C05475=1188.740,321.478,-72.281,-176.478,7.828,148.484
C05476=1188.743,321.230,-72.249,-176.480,7.825,148.484
C05477=1188.748,320.982,-72.218,-176.482,7.823,148.484
C05478=1188.752,320.734,-72.187,-176.485,7.820,148.484
C05479=1188.756,320.486,-72.156,-176.487,7.816,148.484
C05480=1188.760,320.238,-72.124,-176.490,7.813,148.484
C05481=1188.765,319.990,-72.093,-176.492,7.810,148.484
C05482=1188.769,319.743,-72.062,-176.495,7.807,148.484
C05483=1188.773,319.494,-72.031,-176.497,7.805,148.484
C05484=1188.777,319.246,-72.000,-176.499,7.802,148.484
C05485=1188.780,318.999,-71.969,-176.502,7.799,148.484
C05486=1188.785,318.751,-71.938,-176.504,7.795,148.484
C05487=1188.789,318.503,-71.906,-176.507,7.792,148.484
C05488=1188.793,318.255,-71.875,-176.509,7.789,148.484
C05489=1188.797,318.006,-71.844,-176.512,7.786,148.483
C05490=1188.802,317.759,-71.813,-176.514,7.784,148.483
C05491=1188.806,317.511,-71.782,-176.516,7.781,148.483
C05492=1188.810,317.262,-71.751,-176.519,7.777,148.483
C05493=1188.815,317.014,-71.720,-176.521,7.774,148.483
C05494=1188.819,316.766,-71.688,-176.524,7.771,148.483
C05495=1188.823,316.518,-71.657,-176.526,7.768,148.483
C05496=1188.827,316.271,-71.627,-176.529,7.766,148.483
C05497=1188.831,316.022,-71.596,-176.531,7.763,148.483
C05498=1188.835,315.775,-71.565,-176.533,7.759,148.483
C05499=1188.840,315.527,-71.534,-176.536,7.756,148.483
C05500=1188.844,315.278,-71.503,-176.539,7.753,148.483
C05501=1188.849,315.030,-71.472,-176.541,7.750,148.483
C05502=1188.853,314.753,-71.437,-176.544,7.747,148.483
C05503=1188.858,314.477,-71.404,-176.547,7.744,148.483
C05504=1188.862,314.201,-71.369,-176.549,7.741,148.483
C05505=1188.867,313.924,-71.334,-176.553,7.737,148.483
C05506=1188.871,313.676,-71.304,-176.554,7.735,148.483
C05507=1188.876,313.428,-71.273,-176.557,7.732,148.483
C05508=1188.880,313.180,-71.242,-176.560,7.729,148.483
C05509=1188.884,312.932,-71.211,-176.562,7.725,148.482
C05510=1188.888,312.684,-71.181,-176.565,7.722,148.482
C05511=1188.893,312.436,-71.150,-176.567,7.719,148.482
C05512=1188.897,312.187,-71.119,-176.569,7.717,148.482
C05513=1188.901,311.939,-71.088,-176.572,7.714,148.482
C05514=1188.905,311.692,-71.058,-176.574,7.711,148.482
C05515=1188.909,311.443,-71.027,-176.577,7.708,148.482
C05516=1188.914,311.195,-70.996,-176.579,7.705,148.482
C05517=1188.918,310.947,-70.966,-176.581,7.702,148.482
C05518=1188.922,310.699,-70.935,-176.584,7.699,148.482
C05519=1188.926,310.451,-70.904,-176.587,7.696,148.482
C05520=1188.930,310.203,-70.874,-176.589,7.693,148.482
C05521=1188.935,309.955,-70.843,-176.592,7.690,148.482
C05522=1188.939,309.707,-70.812,-176.594,7.688,148.482
C05523=1188.943,309.459,-70.782,-176.597,7.685,148.482
C05524=1188.948,309.210,-70.752,-176.599,7.682,148.482
C05525=1188.952,308.962,-70.721,-176.602,7.679,148.482
C05526=1188.956,308.715,-70.691,-176.604,7.676,148.482
C05527=1188.960,308.466,-70.660,-176.607,7.673,148.482
C05528=1188.964,308.218,-70.630,-176.609,7.670,148.482
C05529=1188.969,307.970,-70.599,-176.611,7.667,148.482
C05530=1188.973,307.722,-70.569,-176.614,7.664,148.482
C05531=1188.977,307.474,-70.539,-176.617,7.661,148.482
C05532=1188.981,307.226,-70.507,-176.620,7.658,148.482
C05533=1188.985,306.978,-70.477,-176.622,7.656,148.482
C05534=1188.990,306.729,-70.447,-176.624,7.653,148.482
C05535=1188.995,306.481,-70.416,-176.627,7.650,148.482
C05536=1188.999,306.234,-70.386,-176.629,7.647,148.482
C05537=1189.003,305.986,-70.356,-176.632,7.644,148.482
C05538=1189.007,305.737,-70.326,-176.634,7.641,148.482
C05539=1189.011,305.489,-70.295,-176.637,7.638,148.482
C05540=1189.015,305.241,-70.265,-176.639,7.635,148.482
C05541=1189.020,304.993,-70.235,-176.642,7.632,148.482
C05542=1189.024,304.745,-70.205,-176.644,7.630,148.482
C05543=1189.029,304.496,-70.175,-176.647,7.627,148.482
C05544=1189.032,304.248,-70.144,-176.649,7.624,148.482
C05545=1189.037,304.000,-70.113,-176.652,7.621,148.482
C05546=1189.041,303.752,-70.084,-176.654,7.618,148.482
C05547=1189.045,303.504,-70.054,-176.657,7.615,148.482
C05548=1189.050,303.256,-70.024,-176.659,7.612,148.482
C05549=1189.054,303.008,-69.993,-176.662,7.609,148.482
C05550=1189.059,302.759,-69.963,-176.665,7.606,148.482
C05551=1189.063,302.512,-69.933,-176.667,7.604,148.482
C05552=1189.068,302.263,-69.903,-176.669,7.601,148.482
C05553=1189.071,302.015,-69.873,-176.672,7.598,148.482
C05554=1189.075,301.767,-69.843,-176.675,7.595,148.482
C05555=1189.080,301.519,-69.812,-176.677,7.592,148.482
C05556=1189.084,301.270,-69.783,-176.679,7.590,148.482
C05557=1189.088,301.023,-69.753,-176.682,7.587,148.482
C05558=1189.093,300.774,-69.723,-176.685,7.584,148.482
C05559=1189.096,300.526,-69.693,-176.688,7.581,148.482
C05560=1189.101,300.278,-69.662,-176.689,7.578,148.482
C05561=1189.106,300.030,-69.633,-176.692,7.575,148.482
C05562=1189.109,299.782,-69.603,-176.695,7.572,148.482
C05563=1189.114,299.534,-69.573,-176.697,7.569,148.482
C05564=1189.118,299.286,-69.543,-176.700,7.567,148.482
C05565=1189.122,299.037,-69.513,-176.702,7.564,148.482
C05566=1189.127,298.789,-69.484,-176.705,7.561,148.482
C05567=1189.131,298.541,-69.453,-176.708,7.558,148.482
C05568=1189.135,298.293,-69.424,-176.710,7.555,148.482
C05569=1189.140,298.045,-69.394,-176.712,7.552,148.482
C05570=1189.144,297.796,-69.365,-176.715,7.549,148.482
C05571=1189.148,297.548,-69.334,-176.717,7.546,148.482
C05572=1189.153,297.300,-69.304,-176.720,7.543,148.482
C05573=1189.157,297.052,-69.275,-176.722,7.541,148.482
C05574=1189.161,296.804,-69.245,-176.725,7.538,148.482
C05575=1189.165,296.556,-69.215,-176.728,7.535,148.482
C05576=1189.170,296.307,-69.185,-176.730,7.532,148.482
C05577=1189.174,296.059,-69.156,-176.733,7.530,148.482
C05578=1189.178,295.811,-69.126,-176.735,7.527,148.482
C05579=1189.182,295.563,-69.097,-176.738,7.524,148.482
C05580=1189.186,295.315,-69.067,-176.740,7.522,148.482
C05581=1189.191,295.066,-69.037,-176.743,7.519,148.482
C05582=1189.195,294.818,-69.007,-176.746,7.516,148.482
C05583=1189.199,294.570,-68.978,-176.748,7.513,148.482
C05584=1189.204,294.322,-68.948,-176.750,7.510,148.482
C05585=1189.208,294.073,-68.919,-176.753,7.507,148.482
C05586=1189.212,293.825,-68.889,-176.755,7.504,148.482
C05587=1189.216,293.577,-68.860,-176.758,7.501,148.482
C05588=1189.220,293.329,-68.831,-176.760,7.499,148.482
C05589=1189.225,293.080,-68.800,-176.763,7.496,148.482
C05590=1189.229,292.832,-68.771,-176.766,7.493,148.482
C05591=1189.234,292.583,-68.742,-176.768,7.490,148.482
C05592=1189.238,292.336,-68.712,-176.771,7.488,148.482
C05593=1189.243,292.088,-68.683,-176.773,7.485,148.482
C05594=1189.247,291.839,-68.654,-176.776,7.482,148.482
C05595=1189.251,291.591,-68.624,-176.778,7.480,148.482
C05596=1189.255,291.343,-68.595,-176.781,7.477,148.482
C05597=1189.259,291.094,-68.565,-176.784,7.474,148.482
C05598=1189.263,290.846,-68.536,-176.786,7.471,148.482
C05599=1189.268,290.598,-68.506,-176.788,7.469,148.483
C05600=1189.272,290.350,-68.477,-176.791,7.466,148.483
C05601=1189.277,290.102,-68.448,-176.794,7.463,148.483
C05602=1189.281,289.854,-68.418,-176.796,7.461,148.483
C05603=1189.285,289.605,-68.390,-176.799,7.458,148.483
C05604=1189.289,289.357,-68.360,-176.801,7.455,148.483
C05605=1189.294,289.108,-68.331,-176.804,7.452,148.483
C05606=1189.298,288.835,-68.298,-176.807,7.449,148.483
C05607=1189.303,288.559,-68.266,-176.810,7.446,148.483
C05608=1189.308,288.285,-68.234,-176.812,7.443,148.483
C05609=1189.313,288.011,-68.201,-176.815,7.440,148.483
C05610=1189.318,287.762,-68.172,-176.818,7.437,148.483
C05611=1189.321,287.514,-68.144,-176.820,7.435,148.483
C05612=1189.325,287.266,-68.114,-176.823,7.432,148.483
C05613=1189.330,287.018,-68.085,-176.826,7.429,148.483
C05614=1189.334,286.769,-68.056,-176.828,7.427,148.483
C05615=1189.339,286.521,-68.027,-176.831,7.424,148.483
C05616=1189.343,286.273,-67.997,-176.833,7.421,148.483
C05617=1189.347,286.024,-67.969,-176.836,7.418,148.483
C05618=1189.352,285.776,-67.940,-176.838,7.415,148.483
C05619=1189.356,285.528,-67.911,-176.841,7.412,148.483
C05620=1189.360,285.280,-67.882,-176.844,7.409,148.483
C05621=1189.364,285.031,-67.852,-176.846,7.407,148.484
C05622=1189.369,284.784,-67.823,-176.849,7.404,148.484
C05623=1189.374,284.535,-67.795,-176.851,7.401,148.484
C05624=1189.378,284.287,-67.765,-176.853,7.399,148.484
C05625=1189.381,284.038,-67.737,-176.856,7.396,148.484
C05626=1189.386,283.790,-67.708,-176.859,7.393,148.484
C05627=1189.391,283.541,-67.679,-176.861,7.391,148.484
C05628=1189.395,283.293,-67.650,-176.864,7.388,148.484
C05629=1189.399,283.044,-67.621,-176.866,7.385,148.484
C05630=1189.403,282.797,-67.593,-176.869,7.383,148.484
C05631=1189.408,282.548,-67.564,-176.872,7.380,148.484
C05632=1189.412,282.300,-67.534,-176.874,7.377,148.484
C05633=1189.417,282.052,-67.506,-176.877,7.375,148.484
C05634=1189.421,281.804,-67.477,-176.879,7.372,148.484
C05635=1189.425,281.555,-67.448,-176.882,7.369,148.484
C05636=1189.430,281.307,-67.419,-176.884,7.367,148.484
C05637=1189.434,281.059,-67.391,-176.887,7.364,148.485
C05638=1189.438,280.810,-67.362,-176.890,7.361,148.485
C05639=1189.443,280.562,-67.333,-176.892,7.359,148.485
C05640=1189.447,280.314,-67.305,-176.895,7.356,148.485
C05641=1189.451,280.065,-67.276,-176.898,7.353,148.485
C05642=1189.456,279.817,-67.247,-176.900,7.351,148.485
C05643=1189.460,279.569,-67.219,-176.903,7.348,148.485
C05644=1189.464,279.320,-67.190,-176.905,7.345,148.485
C05645=1189.469,279.072,-67.161,-176.907,7.343,148.485
C05646=1189.473,278.824,-67.133,-176.910,7.340,148.485
C05647=1189.477,278.575,-67.104,-176.913,7.337,148.485
C05648=1189.482,278.327,-67.075,-176.915,7.334,148.485
C05649=1189.486,278.079,-67.047,-176.918,7.331,148.485
C05650=1189.490,277.831,-67.018,-176.920,7.330,148.486
C05651=1189.494,277.582,-66.990,-176.923,7.327,148.486
C05652=1189.499,277.334,-66.961,-176.926,7.324,148.486
C05653=1189.503,277.086,-66.934,-176.928,7.321,148.486
C05654=1189.508,276.837,-66.905,-176.931,7.318,148.486
C05655=1189.512,276.589,-66.876,-176.933,7.315,148.486
C05656=1189.516,276.341,-66.848,-176.936,7.313,148.486
C05657=1189.521,276.092,-66.819,-176.938,7.310,148.486
C05658=1189.525,275.844,-66.791,-176.941,7.308,148.486
C05659=1189.529,275.595,-66.762,-176.944,7.305,148.486
C05660=1189.534,275.347,-66.735,-176.946,7.302,148.486
C05661=1189.538,275.099,-66.705,-176.948,7.300,148.486
C05662=1189.542,274.851,-66.677,-176.951,7.297,148.486
C05663=1189.547,274.602,-66.649,-176.954,7.294,148.487
C05664=1189.551,274.354,-66.620,-176.956,7.292,148.487
C05665=1189.556,274.105,-66.592,-176.959,7.289,148.487
C05666=1189.559,273.857,-66.564,-176.962,7.286,148.487
C05667=1189.564,273.609,-66.536,-176.964,7.284,148.487
C05668=1189.568,273.360,-66.507,-176.967,7.281,148.487
C05669=1189.573,273.112,-66.480,-176.969,7.279,148.487
C05670=1189.577,272.863,-66.451,-176.972,7.276,148.487
C05671=1189.581,272.615,-66.423,-176.975,7.273,148.487
C05672=1189.586,272.367,-66.394,-176.977,7.271,148.487
C05673=1189.590,272.119,-66.367,-176.980,7.268,148.488
C05674=1189.594,271.870,-66.338,-176.982,7.266,148.488
C05675=1189.599,271.622,-66.310,-176.985,7.263,148.488
C05676=1189.603,271.373,-66.282,-176.988,7.260,148.488
C05677=1189.608,271.125,-66.254,-176.990,7.258,148.488
C05678=1189.612,270.877,-66.225,-176.993,7.255,148.488
C05679=1189.616,270.629,-66.198,-176.995,7.253,148.488
C05680=1189.621,270.380,-66.169,-176.998,7.250,148.488
C05681=1189.625,270.131,-66.142,-177.000,7.247,148.488
C05682=1189.630,269.883,-66.114,-177.003,7.245,148.488
C05683=1189.634,269.635,-66.085,-177.006,7.242,148.489
C05684=1189.638,269.387,-66.058,-177.008,7.240,148.489
C05685=1189.642,269.138,-66.029,-177.011,7.237,148.489
C05686=1189.647,268.890,-66.001,-177.013,7.235,148.489
C05687=1189.651,268.641,-65.974,-177.016,7.232,148.489
C05688=1189.656,268.393,-65.946,-177.019,7.229,148.489
C05689=1189.661,268.145,-65.917,-177.021,7.227,148.489
C05690=1189.664,267.896,-65.889,-177.024,7.224,148.489
C05691=1189.669,267.648,-65.862,-177.026,7.222,148.489
C05692=1189.673,267.399,-65.834,-177.029,7.219,148.490
C05693=1189.678,267.151,-65.806,-177.031,7.217,148.490
C05694=1189.682,266.903,-65.778,-177.034,7.214,148.490
C05695=1189.686,266.654,-65.751,-177.036,7.211,148.490
C05696=1189.691,266.406,-65.723,-177.039,7.209,148.490
C05697=1189.694,266.157,-65.695,-177.042,7.206,148.490
C05698=1189.700,265.908,-65.667,-177.044,7.204,148.490
C05699=1189.704,265.661,-65.639,-177.047,7.201,148.490
C05700=1189.708,265.412,-65.611,-177.049,7.199,148.490
C05701=1189.713,265.163,-65.584,-177.052,7.196,148.491
C05702=1189.717,264.916,-65.556,-177.055,7.193,148.491
C05703=1189.722,264.666,-65.528,-177.057,7.191,148.491
C05704=1189.726,264.418,-65.500,-177.060,7.188,148.491
C05705=1189.730,264.170,-65.473,-177.062,7.186,148.491
C05706=1189.735,263.921,-65.445,-177.065,7.183,148.491
C05707=1189.739,263.673,-65.417,-177.067,7.181,148.491
C05708=1189.744,263.425,-65.390,-177.070,7.178,148.491
C05709=1189.747,263.176,-65.362,-177.072,7.176,148.491
C05710=1189.753,262.904,-65.332,-177.075,7.173,148.492
C05711=1189.757,262.630,-65.301,-177.078,7.171,148.492
C05712=1189.762,262.358,-65.271,-177.081,7.168,148.492
C05713=1189.766,262.085,-65.241,-177.084,7.165,148.492
C05714=1189.772,261.836,-65.213,-177.086,7.163,148.492
C05715=1189.776,261.587,-65.186,-177.089,7.160,148.492
C05716=1189.781,261.339,-65.158,-177.091,7.158,148.492
C05717=1189.785,261.090,-65.131,-177.095,7.155,148.493
C05718=1189.789,260.842,-65.103,-177.097,7.152,148.493
C05719=1189.794,260.594,-65.076,-177.099,7.150,148.493
C05720=1189.798,260.345,-65.048,-177.102,7.147,148.493
C05721=1189.802,260.097,-65.021,-177.105,7.145,148.493
C05722=1189.807,259.848,-64.994,-177.108,7.142,148.493
C05723=1189.811,259.600,-64.966,-177.110,7.140,148.493
C05724=1189.815,259.351,-64.939,-177.113,7.137,148.493
C05725=1189.820,259.103,-64.912,-177.115,7.135,148.494
C05726=1189.824,258.855,-64.884,-177.118,7.132,148.494
C05727=1189.829,258.606,-64.857,-177.120,7.130,148.494
C05728=1189.834,258.358,-64.830,-177.123,7.127,148.494
C05729=1189.838,258.109,-64.802,-177.125,7.125,148.494
C05730=1189.842,257.861,-64.774,-177.128,7.122,148.494
C05731=1189.847,257.612,-64.747,-177.131,7.120,148.494
C05732=1189.851,257.364,-64.721,-177.133,7.117,148.494
C05733=1189.855,257.115,-64.693,-177.136,7.115,148.495
C05734=1189.859,256.867,-64.666,-177.139,7.112,148.495
C05735=1189.864,256.619,-64.639,-177.141,7.110,148.495
C05736=1189.868,256.370,-64.612,-177.144,7.107,148.495
C05737=1189.873,256.122,-64.585,-177.146,7.105,148.495
C05738=1189.878,255.873,-64.557,-177.149,7.102,148.495
C05739=1189.881,255.624,-64.529,-177.151,7.100,148.495
C05740=1189.886,255.376,-64.502,-177.154,7.098,148.496
C05741=1189.890,255.128,-64.476,-177.156,7.095,148.496
C05742=1189.895,254.879,-64.449,-177.159,7.092,148.496
C05743=1189.899,254.631,-64.422,-177.162,7.091,148.496
C05744=1189.904,254.382,-64.395,-177.165,7.088,148.496
C05745=1189.908,254.133,-64.367,-177.167,7.086,148.497
C05746=1189.913,253.885,-64.340,-177.170,7.083,148.497
C05747=1189.917,253.636,-64.314,-177.172,7.081,148.497
C05748=1189.921,253.388,-64.287,-177.175,7.079,148.497
C05749=1189.926,253.139,-64.260,-177.177,7.076,148.497
C05750=1189.931,252.891,-64.232,-177.180,7.074,148.497
C05751=1189.935,252.642,-64.205,-177.183,7.071,148.497
C05752=1189.939,252.394,-64.179,-177.185,7.069,148.498
C05753=1189.943,252.145,-64.152,-177.188,7.066,148.498
C05754=1189.948,251.897,-64.124,-177.190,7.064,148.498
C05755=1189.952,251.648,-64.097,-177.193,7.061,148.498
C05756=1189.956,251.400,-64.071,-177.196,7.059,148.498
C05757=1189.961,251.151,-64.044,-177.198,7.056,148.498
C05758=1189.966,250.903,-64.017,-177.201,7.054,148.498
C05759=1189.970,250.655,-63.990,-177.204,7.051,148.499
C05760=1189.974,250.406,-63.963,-177.206,7.049,148.499
C05761=1189.979,250.158,-63.936,-177.208,7.047,148.499
C05762=1189.984,249.909,-63.909,-177.211,7.044,148.499
C05763=1189.988,249.661,-63.883,-177.213,7.042,148.499
C05764=1189.992,249.412,-63.856,-177.217,7.040,148.500
C05765=1189.997,249.163,-63.829,-177.219,7.037,148.500
C05766=1190.001,248.915,-63.803,-177.222,7.034,148.500
C05767=1190.005,248.666,-63.775,-177.224,7.033,148.500
C05768=1190.010,248.418,-63.748,-177.227,7.030,148.500
C05769=1190.014,248.169,-63.723,-177.230,7.028,148.500
C05770=1190.019,247.920,-63.696,-177.232,7.026,148.500
C05771=1190.023,247.672,-63.669,-177.235,7.023,148.501
C05772=1190.027,247.424,-63.642,-177.237,7.021,148.501
C05773=1190.032,247.174,-63.616,-177.240,7.018,148.501
C05774=1190.036,246.926,-63.589,-177.242,7.016,148.501
C05775=1190.041,246.678,-63.562,-177.245,7.013,148.501
C05776=1190.045,246.430,-63.536,-177.248,7.011,148.502
C05777=1190.050,246.180,-63.509,-177.250,7.009,148.502
C05778=1190.054,245.932,-63.482,-177.253,7.006,148.502
C05779=1190.058,245.684,-63.456,-177.255,7.004,148.502
C05780=1190.063,245.435,-63.429,-177.258,7.001,148.502
C05781=1190.067,245.187,-63.403,-177.261,6.999,148.502
C05782=1190.072,244.939,-63.376,-177.263,6.997,148.503
C05783=1190.077,244.690,-63.351,-177.266,6.995,148.503
C05784=1190.081,244.441,-63.323,-177.268,6.992,148.503
C05785=1190.085,244.193,-63.298,-177.271,6.990,148.503
C05786=1190.090,243.944,-63.271,-177.274,6.988,148.503
C05787=1190.094,243.696,-63.244,-177.276,6.985,148.503
C05788=1190.099,243.447,-63.218,-177.279,6.983,148.504
C05789=1190.103,243.199,-63.191,-177.281,6.981,148.504
C05790=1190.108,242.950,-63.165,-177.284,6.978,148.504
C05791=1190.112,242.701,-63.139,-177.286,6.976,148.504
C05792=1190.117,242.452,-63.112,-177.290,6.973,148.504
C05793=1190.121,242.204,-63.086,-177.292,6.971,148.505
C05794=1190.125,241.955,-63.060,-177.294,6.969,148.505
C05795=1190.130,241.707,-63.033,-177.297,6.966,148.505
C05796=1190.134,241.459,-63.008,-177.300,6.964,148.505
C05797=1190.139,241.210,-62.980,-177.302,6.962,148.505
C05798=1190.143,240.961,-62.955,-177.305,6.960,148.506
C05799=1190.148,240.713,-62.928,-177.307,6.957,148.506
C05800=1190.152,240.464,-62.902,-177.311,6.955,148.506
C05801=1190.156,240.215,-62.876,-177.313,6.953,148.506
C05802=1190.161,239.967,-62.849,-177.315,6.951,148.506
C05803=1190.165,239.718,-62.823,-177.318,6.948,148.506
C05804=1190.170,239.470,-62.798,-177.321,6.946,148.507
C05805=1190.175,239.221,-62.771,-177.323,6.944,148.507
C05806=1190.179,238.973,-62.745,-177.326,6.941,148.507
C05807=1190.183,238.724,-62.719,-177.328,6.939,148.507
C05808=1190.188,238.475,-62.692,-177.332,6.936,148.508
C05809=1190.192,238.226,-62.667,-177.334,6.934,148.508
C05810=1190.197,237.978,-62.641,-177.336,6.932,148.508
C05811=1190.202,237.730,-62.614,-177.339,6.929,148.508
C05812=1190.206,237.481,-62.588,-177.342,6.928,148.508
C05813=1190.210,237.232,-62.563,-177.344,6.925,148.508
C05814=1190.214,236.961,-62.534,-177.347,6.923,148.509
C05815=1190.220,236.689,-62.506,-177.350,6.920,148.509
C05816=1190.225,236.418,-62.477,-177.352,6.918,148.509
C05817=1190.230,236.146,-62.449,-177.356,6.915,148.509
C05818=1190.234,235.897,-62.423,-177.358,6.913,148.510
C05819=1190.239,235.649,-62.397,-177.361,6.910,148.510
C05820=1190.243,235.401,-62.371,-177.363,6.908,148.510
C05821=1190.247,235.152,-62.345,-177.366,6.906,148.510
C05822=1190.252,234.903,-62.319,-177.369,6.904,148.511
C05823=1190.256,234.654,-62.293,-177.371,6.902,148.511
C05824=1190.261,234.406,-62.267,-177.374,6.900,148.511
C05825=1190.266,234.157,-62.242,-177.377,6.897,148.511
C05826=1190.270,233.908,-62.216,-177.379,6.895,148.511
C05827=1190.274,233.660,-62.190,-177.381,6.893,148.511
C05828=1190.279,233.412,-62.164,-177.385,6.890,148.512
C05829=1190.284,233.163,-62.138,-177.387,6.888,148.512
C05830=1190.288,232.914,-62.112,-177.389,6.886,148.512
C05831=1190.293,232.666,-62.087,-177.392,6.883,148.512
C05832=1190.297,232.417,-62.061,-177.395,6.881,148.513
C05833=1190.301,232.168,-62.035,-177.397,6.880,148.513
C05834=1190.305,231.920,-62.009,-177.400,6.877,148.513
C05835=1190.310,231.672,-61.984,-177.403,6.875,148.513
C05836=1190.314,231.423,-61.958,-177.405,6.873,148.513
C05837=1190.319,231.174,-61.932,-177.408,6.870,148.514
C05838=1190.324,230.926,-61.906,-177.411,6.868,148.514
C05839=1190.328,230.677,-61.881,-177.413,6.866,148.514
C05840=1190.333,230.428,-61.855,-177.416,6.863,148.514
C05841=1190.338,230.179,-61.830,-177.418,6.861,148.514
C05842=1190.342,229.930,-61.805,-177.421,6.859,148.515
C05843=1190.346,229.682,-61.779,-177.424,6.856,148.515
C05844=1190.351,229.434,-61.753,-177.426,6.855,148.515
C05845=1190.355,229.185,-61.728,-177.429,6.853,148.516
C05846=1190.359,228.936,-61.702,-177.431,6.851,148.516
C05847=1190.364,228.688,-61.676,-177.434,6.848,148.516
C05848=1190.369,228.439,-61.651,-177.437,6.846,148.516
C05849=1190.373,228.190,-61.626,-177.439,6.844,148.516
C05850=1190.378,227.941,-61.600,-177.442,6.841,148.517
C05851=1190.382,227.693,-61.575,-177.445,6.839,148.517
C05852=1190.386,227.444,-61.549,-177.447,6.837,148.517
C05853=1190.391,227.196,-61.523,-177.450,6.835,148.517
C05854=1190.396,226.946,-61.498,-177.453,6.833,148.518
C05855=1190.401,226.698,-61.473,-177.455,6.831,148.518
C05856=1190.405,226.449,-61.447,-177.457,6.829,148.518
C05857=1190.409,226.201,-61.422,-177.461,6.826,148.518
C05858=1190.414,225.952,-61.397,-177.463,6.824,148.519
C05859=1190.418,225.703,-61.371,-177.465,6.822,148.519
C05860=1190.423,225.455,-61.346,-177.469,6.819,148.519
C05861=1190.427,225.206,-61.321,-177.471,6.818,148.519
C05862=1190.431,224.957,-61.296,-177.474,6.815,148.519
C05863=1190.436,224.709,-61.270,-177.476,6.814,148.520
C05864=1190.441,224.460,-61.245,-177.479,6.811,148.520
C05865=1190.445,224.211,-61.220,-177.482,6.809,148.520
C05866=1190.450,223.963,-61.194,-177.484,6.807,148.520
C05867=1190.455,223.714,-61.169,-177.487,6.804,148.521
C05868=1190.459,223.465,-61.144,-177.490,6.802,148.521
C05869=1190.463,223.217,-61.119,-177.492,6.800,148.521
C05870=1190.468,222.968,-61.094,-177.494,6.798,148.521
C05871=1190.472,222.719,-61.068,-177.498,6.796,148.522
C05872=1190.477,222.470,-61.043,-177.500,6.794,148.522
C05873=1190.481,222.222,-61.018,-177.502,6.792,148.522
C05874=1190.486,221.973,-60.993,-177.505,6.790,148.522
C05875=1190.490,221.724,-60.968,-177.508,6.787,148.523
C05876=1190.495,221.476,-60.943,-177.510,6.785,148.523
C05877=1190.499,221.227,-60.917,-177.513,6.783,148.523
C05878=1190.504,220.978,-60.893,-177.516,6.781,148.523
C05879=1190.508,220.729,-60.867,-177.519,6.778,148.524
C05880=1190.513,220.481,-60.843,-177.521,6.777,148.524
C05881=1190.517,220.232,-60.817,-177.524,6.775,148.524
C05882=1190.522,219.983,-60.792,-177.526,6.773,148.524
C05883=1190.526,219.735,-60.767,-177.529,6.770,148.525
C05884=1190.531,219.486,-60.743,-177.532,6.768,148.525
C05885=1190.535,219.237,-60.717,-177.534,6.766,148.525
C05886=1190.540,218.989,-60.692,-177.537,6.764,148.525
C05887=1190.545,218.740,-60.668,-177.540,6.761,148.526
C05888=1190.549,218.491,-60.642,-177.543,6.760,148.526
C05889=1190.554,218.243,-60.618,-177.545,6.758,148.526
C05890=1190.558,217.994,-60.593,-177.547,6.756,148.526
C05891=1190.563,217.745,-60.568,-177.551,6.753,148.527
C05892=1190.567,217.496,-60.543,-177.553,6.751,148.527
C05893=1190.571,217.248,-60.519,-177.555,6.749,148.527
C05894=1190.576,216.999,-60.493,-177.558,6.747,148.528
C05895=1190.581,216.750,-60.468,-177.561,6.745,148.528
C05896=1190.585,216.502,-60.444,-177.563,6.742,148.528
C05897=1190.589,216.253,-60.418,-177.566,6.741,148.528
C05898=1190.595,216.004,-60.394,-177.569,6.739,148.529
C05899=1190.598,215.755,-60.369,-177.571,6.737,148.529
C05900=1190.604,215.506,-60.345,-177.574,6.734,148.529
C05901=1190.608,215.258,-60.321,-177.577,6.732,148.529
C05902=1190.612,215.009,-60.295,-177.579,6.730,148.530
C05903=1190.617,214.760,-60.270,-177.582,6.728,148.530
C05904=1190.621,214.511,-60.246,-177.585,6.726,148.530
C05905=1190.626,214.262,-60.221,-177.587,6.724,148.531
C05906=1190.631,214.014,-60.197,-177.590,6.722,148.531
C05907=1190.635,213.765,-60.171,-177.592,6.720,148.531
C05908=1190.639,213.517,-60.147,-177.595,6.718,148.531
C05909=1190.644,213.268,-60.123,-177.598,6.715,148.532
C05910=1190.648,213.019,-60.098,-177.600,6.713,148.532
C05911=1190.653,212.770,-60.073,-177.603,6.711,148.532
C05912=1190.658,212.522,-60.049,-177.606,6.710,148.532
C05913=1190.662,212.272,-60.024,-177.608,6.708,148.533
C05914=1190.667,212.024,-60.000,-177.611,6.705,148.533
C05915=1190.672,211.775,-59.976,-177.614,6.703,148.533
C05916=1190.676,211.526,-59.951,-177.616,6.701,148.533
C05917=1190.681,211.277,-59.926,-177.619,6.699,148.534
C05918=1190.686,211.007,-59.900,-177.622,6.697,148.534
C05919=1190.691,210.737,-59.873,-177.625,6.695,148.534
C05920=1190.695,210.467,-59.847,-177.628,6.692,148.535
C05921=1190.700,210.196,-59.820,-177.630,6.690,148.535
C05922=1190.705,209.948,-59.795,-177.633,6.688,148.535
C05923=1190.709,209.699,-59.771,-177.636,6.686,148.536
C05924=1190.714,209.450,-59.746,-177.639,6.684,148.536
C05925=1190.718,209.201,-59.722,-177.641,6.682,148.536
C05926=1190.723,208.952,-59.699,-177.644,6.680,148.536
C05927=1190.728,208.703,-59.674,-177.646,6.678,148.537
C05928=1190.732,208.455,-59.649,-177.649,6.676,148.537
C05929=1190.737,208.206,-59.625,-177.652,6.674,148.537
C05930=1190.742,207.957,-59.601,-177.654,6.672,148.537
C05931=1190.745,207.708,-59.576,-177.657,6.670,148.538
C05932=1190.750,207.460,-59.552,-177.660,6.668,148.538
C05933=1190.755,207.211,-59.528,-177.662,6.666,148.538
C05934=1190.759,206.963,-59.503,-177.664,6.664,148.539
C05935=1190.764,206.713,-59.479,-177.668,6.661,148.539
C05936=1190.768,206.464,-59.455,-177.670,6.660,148.539
C05937=1190.773,206.216,-59.431,-177.673,6.658,148.540
C05938=1190.778,205.967,-59.406,-177.676,6.656,148.540
C05939=1190.782,205.719,-59.382,-177.678,6.654,148.540
C05940=1190.786,205.469,-59.359,-177.681,6.652,148.540
C05941=1190.792,205.220,-59.334,-177.684,6.649,148.541
C05942=1190.796,204.972,-59.310,-177.686,6.648,148.541
C05943=1190.800,204.724,-59.286,-177.689,6.646,148.541
C05944=1190.805,204.474,-59.262,-177.691,6.644,148.542
C05945=1190.810,204.225,-59.237,-177.694,6.642,148.542
C05946=1190.814,203.977,-59.213,-177.697,6.640,148.542
C05947=1190.819,203.728,-59.190,-177.699,6.638,148.543
C05948=1190.823,203.479,-59.166,-177.702,6.636,148.543
C05949=1190.828,203.230,-59.141,-177.705,6.633,148.543
C05950=1190.833,202.981,-59.118,-177.707,6.632,148.543
C05951=1190.837,202.733,-59.094,-177.710,6.630,148.544
C05952=1190.841,202.484,-59.069,-177.713,6.628,148.544
C05953=1190.846,202.235,-59.046,-177.715,6.626,148.544
C05954=1190.851,201.986,-59.021,-177.718,6.624,148.545
C05955=1190.856,201.737,-58.998,-177.721,6.621,148.545
C05956=1190.860,201.489,-58.974,-177.723,6.620,148.545
C05957=1190.864,201.240,-58.950,-177.726,6.618,148.545
C05958=1190.869,200.991,-58.926,-177.729,6.616,148.546
C05959=1190.873,200.742,-58.902,-177.731,6.614,148.546
C05960=1190.878,200.493,-58.878,-177.734,6.612,148.547
C05961=1190.883,200.244,-58.854,-177.736,6.610,148.547
C05962=1190.887,199.995,-58.831,-177.739,6.608,148.547
C05963=1190.892,199.747,-58.806,-177.742,6.606,148.547
C05964=1190.897,199.498,-58.783,-177.745,6.604,148.548
C05965=1190.901,199.250,-58.759,-177.747,6.602,148.548
C05966=1190.906,199.000,-58.736,-177.750,6.600,148.548
C05967=1190.910,198.752,-58.712,-177.752,6.598,148.548
C05968=1190.915,198.503,-58.688,-177.755,6.596,148.549
C05969=1190.920,198.254,-58.664,-177.757,6.595,148.549
C05970=1190.925,198.005,-58.640,-177.760,6.593,148.550
C05971=1190.929,197.756,-58.617,-177.763,6.591,148.550
C05972=1190.933,197.507,-58.592,-177.766,6.588,148.550
C05973=1190.938,197.258,-58.569,-177.768,6.586,148.550
C05974=1190.942,197.010,-58.545,-177.771,6.584,148.551
C05975=1190.947,196.761,-58.522,-177.774,6.583,148.551
C05976=1190.952,196.512,-58.498,-177.776,6.581,148.551
C05977=1190.956,196.263,-58.474,-177.779,6.579,148.552
C05978=1190.961,196.014,-58.451,-177.781,6.577,148.552
C05979=1190.965,195.765,-58.427,-177.784,6.575,148.552
C05980=1190.970,195.517,-58.403,-177.787,6.574,148.553
C05981=1190.974,195.268,-58.380,-177.789,6.572,148.553
C05982=1190.979,195.019,-58.357,-177.792,6.570,148.553
C05983=1190.984,194.770,-58.333,-177.795,6.567,148.554
C05984=1190.988,194.521,-58.309,-177.798,6.565,148.554
C05985=1190.993,194.272,-58.286,-177.800,6.563,148.554
C05986=1190.998,194.023,-58.263,-177.803,6.562,148.555
C05987=1191.002,193.775,-58.238,-177.806,6.560,148.555
C05988=1191.007,193.526,-58.215,-177.808,6.558,148.555
C05989=1191.011,193.277,-58.192,-177.810,6.556,148.555
C05990=1191.015,193.028,-58.169,-177.813,6.554,148.556
C05991=1191.020,192.779,-58.146,-177.816,6.552,148.556
C05992=1191.025,192.531,-58.122,-177.818,6.551,148.556
C05993=1191.029,192.281,-58.098,-177.821,6.549,148.557
C05994=1191.035,192.033,-58.075,-177.824,6.547,148.557
C05995=1191.039,191.784,-58.052,-177.826,6.545,148.558
C05996=1191.044,191.535,-58.028,-177.830,6.543,148.558
C05997=1191.049,191.286,-58.005,-177.832,6.541,148.558
C05998=1191.053,191.037,-57.982,-177.834,6.539,148.558
C05999=1191.057,190.789,-57.958,-177.837,6.537,148.559
C06000=1191.062,190.540,-57.935,-177.840,6.535,148.559
C06001=1191.066,190.291,-57.912,-177.842,6.533,148.559
C06002=1191.071,190.042,-57.888,-177.845,6.531,148.560
C06003=1191.076,189.793,-57.865,-177.848,6.530,148.560
C06004=1191.080,189.544,-57.841,-177.850,6.528,148.560
C06005=1191.085,189.296,-57.819,-177.853,6.526,148.561
C06006=1191.090,189.047,-57.796,-177.856,6.524,148.561
C06007=1191.094,188.798,-57.772,-177.858,6.522,148.561
C06008=1191.099,188.549,-57.749,-177.861,6.521,148.562
C06009=1191.104,188.300,-57.726,-177.863,6.518,148.562
C06010=1191.108,188.051,-57.703,-177.866,6.517,148.562
C06011=1191.112,187.802,-57.680,-177.869,6.515,148.563
C06012=1191.117,187.553,-57.656,-177.871,6.513,148.563
C06013=1191.122,187.304,-57.633,-177.874,6.511,148.563
C06014=1191.126,187.056,-57.610,-177.877,6.509,148.564
C06015=1191.131,186.807,-57.587,-177.879,6.508,148.564
C06016=1191.136,186.558,-57.564,-177.882,6.506,148.564
C06017=1191.140,186.308,-57.542,-177.885,6.504,148.565
C06018=1191.145,186.059,-57.518,-177.887,6.502,148.565
C06019=1191.150,185.810,-57.495,-177.890,6.500,148.566
C06020=1191.155,185.562,-57.472,-177.893,6.499,148.566
C06021=1191.159,185.313,-57.449,-177.896,6.496,148.566
C06022=1191.164,185.043,-57.424,-177.898,6.494,148.567
C06023=1191.169,184.774,-57.400,-177.901,6.492,148.567
C06024=1191.174,184.504,-57.375,-177.904,6.491,148.567
C06025=1191.179,184.234,-57.350,-177.907,6.488,148.568
C06026=1191.183,183.986,-57.327,-177.910,6.486,148.568
C06027=1191.188,183.737,-57.304,-177.912,6.484,148.568
C06028=1191.193,183.488,-57.280,-177.915,6.483,148.569
C06029=1191.198,183.239,-57.258,-177.918,6.481,148.569
C06030=1191.202,182.990,-57.235,-177.920,6.479,148.569
C06031=1191.206,182.741,-57.212,-177.923,6.477,148.570
C06032=1191.211,182.492,-57.189,-177.926,6.475,148.570
C06033=1191.217,182.243,-57.167,-177.928,6.474,148.570
C06034=1191.220,181.995,-57.144,-177.931,6.472,148.571
C06035=1191.225,181.746,-57.121,-177.934,6.470,148.571
C06036=1191.229,181.496,-57.099,-177.936,6.468,148.571
C06037=1191.235,181.248,-57.076,-177.939,6.467,148.572
C06038=1191.239,180.999,-57.053,-177.942,6.465,148.572
C06039=1191.244,180.750,-57.030,-177.944,6.463,148.573
C06040=1191.248,180.500,-57.007,-177.947,6.461,148.573
C06041=1191.253,180.252,-56.984,-177.949,6.459,148.573
C06042=1191.258,180.003,-56.962,-177.952,6.457,148.573
C06043=1191.262,179.754,-56.939,-177.954,6.456,148.574
C06044=1191.267,179.505,-56.916,-177.957,6.454,148.574
C06045=1191.272,179.256,-56.894,-177.959,6.453,148.575
C06046=1191.276,179.007,-56.871,-177.962,6.451,148.575
C06047=1191.280,178.758,-56.849,-177.965,6.449,148.575
C06048=1191.286,178.510,-56.826,-177.967,6.447,148.576
C06049=1191.290,178.260,-56.803,-177.970,6.445,148.576
C06050=1191.295,178.011,-56.780,-177.973,6.444,148.576
C06051=1191.300,177.763,-56.758,-177.975,6.442,148.577
C06052=1191.304,177.514,-56.736,-177.978,6.440,148.577
C06053=1191.309,177.264,-56.713,-177.981,6.438,148.577
C06054=1191.313,177.016,-56.691,-177.983,6.437,148.578
C06055=1191.318,176.767,-56.668,-177.986,6.435,148.578
C06056=1191.322,176.518,-56.645,-177.989,6.433,148.578
C06057=1191.328,176.269,-56.623,-177.991,6.431,148.579
C06058=1191.332,176.020,-56.600,-177.994,6.429,148.579
C06059=1191.336,175.771,-56.578,-177.997,6.428,148.580
C06060=1191.341,175.523,-56.555,-177.999,6.426,148.580
C06061=1191.346,175.273,-56.533,-178.002,6.424,148.580
C06062=1191.351,175.024,-56.510,-178.005,6.422,148.581
C06063=1191.355,174.776,-56.488,-178.007,6.420,148.581
C06064=1191.359,174.526,-56.466,-178.010,6.419,148.581
C06065=1191.365,174.278,-56.443,-178.013,6.417,148.582
C06066=1191.369,174.029,-56.421,-178.015,6.415,148.582
C06067=1191.373,173.779,-56.399,-178.018,6.413,148.582
C06068=1191.379,173.531,-56.376,-178.020,6.412,148.583
C06069=1191.383,173.282,-56.354,-178.023,6.410,148.583
C06070=1191.388,173.033,-56.332,-178.026,6.409,148.584
C06071=1191.392,172.784,-56.309,-178.029,6.407,148.584
C06072=1191.397,172.535,-56.287,-178.031,6.405,148.585
C06073=1191.401,172.286,-56.265,-178.034,6.404,148.585
C06074=1191.406,172.036,-56.242,-178.037,6.402,148.585
C06075=1191.411,171.788,-56.220,-178.039,6.400,148.586
C06076=1191.415,171.539,-56.198,-178.042,6.398,148.586
C06077=1191.420,171.290,-56.176,-178.045,6.397,148.586
C06078=1191.425,171.041,-56.154,-178.047,6.395,148.587
C06079=1191.429,170.792,-56.131,-178.050,6.393,148.587
C06080=1191.434,170.543,-56.109,-178.053,6.391,148.587
C06081=1191.438,170.294,-56.087,-178.055,6.389,148.588
C06082=1191.444,170.045,-56.065,-178.058,6.388,148.588
C06083=1191.448,169.796,-56.043,-178.060,6.387,148.589
C06084=1191.453,169.548,-56.020,-178.063,6.385,148.589
C06085=1191.457,169.298,-55.998,-178.066,6.383,148.589
C06086=1191.463,169.049,-55.976,-178.068,6.381,148.590
C06087=1191.467,168.800,-55.954,-178.071,6.379,148.590
C06088=1191.472,168.551,-55.932,-178.074,6.378,148.590
C06089=1191.476,168.302,-55.910,-178.076,6.376,148.591
C06090=1191.481,168.053,-55.889,-178.079,6.374,148.591
C06091=1191.485,167.804,-55.867,-178.082,6.372,148.591
C06092=1191.491,167.555,-55.844,-178.084,6.372,148.592
C06093=1191.495,167.306,-55.822,-178.087,6.370,148.592
C06094=1191.500,167.058,-55.800,-178.090,6.368,148.593
C06095=1191.504,166.808,-55.778,-178.092,6.366,148.593
C06096=1191.509,166.560,-55.756,-178.095,6.365,148.594
C06097=1191.513,166.310,-55.734,-178.098,6.363,148.594
C06098=1191.518,166.062,-55.712,-178.100,6.361,148.594
C06099=1191.522,165.812,-55.690,-178.103,6.359,148.595
C06100=1191.528,165.563,-55.668,-178.106,6.357,148.595
C06101=1191.533,165.315,-55.646,-178.108,6.356,148.595
C06102=1191.537,165.065,-55.624,-178.110,6.355,148.596
C06103=1191.542,164.817,-55.603,-178.113,6.353,148.596
C06104=1191.546,164.567,-55.581,-178.116,6.351,148.597
C06105=1191.551,164.318,-55.560,-178.118,6.349,148.597
C06106=1191.555,164.069,-55.538,-178.122,6.348,148.597
C06107=1191.560,163.820,-55.516,-178.124,6.346,148.598
C06108=1191.565,163.572,-55.494,-178.127,6.344,148.598
C06109=1191.569,163.322,-55.472,-178.129,6.343,148.599
C06110=1191.574,163.074,-55.451,-178.132,6.342,148.599
C06111=1191.579,162.824,-55.429,-178.134,6.340,148.599
C06112=1191.583,162.576,-55.407,-178.137,6.338,148.600
C06113=1191.588,162.327,-55.385,-178.140,6.336,148.600
C06114=1191.593,162.077,-55.364,-178.142,6.334,148.600
C06115=1191.598,161.828,-55.342,-178.145,6.333,148.601
C06116=1191.602,161.579,-55.320,-178.148,6.331,148.601
C06117=1191.607,161.330,-55.298,-178.150,6.330,148.602
C06118=1191.612,161.082,-55.277,-178.153,6.329,148.602
C06119=1191.616,160.832,-55.255,-178.156,6.327,148.603
C06120=1191.621,160.583,-55.234,-178.158,6.325,148.603
C06121=1191.626,160.335,-55.212,-178.161,6.323,148.603
C06122=1191.630,160.085,-55.190,-178.164,6.321,148.604
C06123=1191.636,159.836,-55.169,-178.166,6.320,148.604
C06124=1191.640,159.587,-55.147,-178.169,6.319,148.604
C06125=1191.645,159.338,-55.125,-178.171,6.317,148.605
C06126=1191.649,159.069,-55.103,-178.174,6.315,148.605
C06127=1191.655,158.800,-55.078,-178.177,6.314,148.606
C06128=1191.659,158.531,-55.056,-178.180,6.312,148.606
C06129=1191.665,158.262,-55.032,-178.183,6.310,148.607
C06130=1191.670,158.013,-55.011,-178.186,6.309,148.607
C06131=1191.674,157.764,-54.990,-178.188,6.307,148.607
C06132=1191.678,157.515,-54.968,-178.191,6.305,148.608
C06133=1191.683,157.266,-54.947,-178.194,6.303,148.608
C06134=1191.688,157.017,-54.926,-178.196,6.302,148.609
C06135=1191.693,156.768,-54.904,-178.198,6.301,148.609
C06136=1191.698,156.518,-54.883,-178.202,6.299,148.610
C06137=1191.703,156.270,-54.861,-178.204,6.297,148.610
C06138=1191.707,156.021,-54.840,-178.207,6.296,148.610
C06139=1191.711,155.771,-54.818,-178.210,6.294,148.611
C06140=1191.716,155.523,-54.797,-178.212,6.292,148.611
C06141=1191.722,155.273,-54.776,-178.214,6.291,148.611
C06142=1191.726,155.025,-54.754,-178.217,6.289,148.612
C06143=1191.730,154.775,-54.733,-178.220,6.288,148.612
C06144=1191.735,154.527,-54.712,-178.223,6.286,148.613
C06145=1191.740,154.277,-54.691,-178.226,6.284,148.613
C06146=1191.745,154.029,-54.669,-178.228,6.283,148.614
C06147=1191.750,153.779,-54.648,-178.230,6.282,148.614
C06148=1191.754,153.530,-54.627,-178.233,6.280,148.614
C06149=1191.759,153.281,-54.606,-178.236,6.278,148.615
C06150=1191.764,153.032,-54.584,-178.239,6.277,148.615
C06151=1191.769,152.783,-54.563,-178.241,6.276,148.616
C06152=1191.773,152.534,-54.542,-178.244,6.274,148.616
C06153=1191.778,152.285,-54.521,-178.246,6.272,148.616
C06154=1191.783,152.036,-54.500,-178.249,6.270,148.617
C06155=1191.787,151.787,-54.479,-178.252,6.269,148.617
C06156=1191.792,151.538,-54.458,-178.254,6.268,148.618
C06157=1191.797,151.289,-54.436,-178.257,6.266,148.618
C06158=1191.802,151.039,-54.415,-178.260,6.264,148.619
C06159=1191.806,150.790,-54.394,-178.262,6.263,148.619
C06160=1191.811,150.542,-54.373,-178.265,6.261,148.619
C06161=1191.816,150.293,-54.352,-178.267,6.260,148.620
C06162=1191.820,150.043,-54.331,-178.270,6.258,148.620
C06163=1191.825,149.794,-54.309,-178.273,6.257,148.621
C06164=1191.829,149.545,-54.289,-178.276,6.255,148.621
C06165=1191.834,149.296,-54.268,-178.278,6.254,148.622
C06166=1191.839,149.047,-54.246,-178.281,6.252,148.622
C06167=1191.844,148.799,-54.226,-178.284,6.251,148.623
C06168=1191.849,148.549,-54.205,-178.286,6.249,148.623
C06169=1191.854,148.299,-54.183,-178.288,6.248,148.623
C06170=1191.858,148.051,-54.162,-178.291,6.246,148.624
C06171=1191.863,147.802,-54.141,-178.294,6.244,148.624
C06172=1191.867,147.553,-54.121,-178.297,6.243,148.625
C06173=1191.872,147.303,-54.100,-178.300,6.241,148.625
C06174=1191.877,147.055,-54.080,-178.302,6.240,148.625
C06175=1191.882,146.806,-54.058,-178.304,6.239,148.626
C06176=1191.887,146.557,-54.037,-178.307,6.237,148.626
C06177=1191.891,146.308,-54.017,-178.310,6.235,148.627
C06178=1191.896,146.058,-53.995,-178.312,6.234,148.627
C06179=1191.900,145.809,-53.975,-178.315,6.233,148.628
C06180=1191.906,145.560,-53.954,-178.318,6.231,148.628
C06181=1191.910,145.311,-53.933,-178.321,6.229,148.628
C06182=1191.915,145.062,-53.912,-178.323,6.228,148.629
C06183=1191.919,144.813,-53.892,-178.326,6.227,148.629
C06184=1191.924,144.564,-53.871,-178.328,6.225,148.630
C06185=1191.929,144.315,-53.850,-178.331,6.223,148.630
C06186=1191.934,144.066,-53.829,-178.333,6.222,148.630
C06187=1191.939,143.817,-53.809,-178.336,6.221,148.631
C06188=1191.944,143.567,-53.788,-178.339,6.219,148.631
C06189=1191.948,143.318,-53.768,-178.342,6.217,148.632
C06190=1191.953,143.069,-53.747,-178.344,6.216,148.632
C06191=1191.958,142.820,-53.726,-178.347,6.215,148.633
C06192=1191.962,142.571,-53.705,-178.350,6.213,148.633
C06193=1191.967,142.321,-53.684,-178.352,6.212,148.634
C06194=1191.971,142.072,-53.664,-178.355,6.210,148.634
C06195=1191.976,141.823,-53.643,-178.357,6.209,148.634
C06196=1191.981,141.574,-53.623,-178.360,6.207,148.635
C06197=1191.985,141.325,-53.602,-178.363,6.206,148.635
C06198=1191.990,141.076,-53.581,-178.365,6.205,148.636
C06199=1191.995,140.827,-53.561,-178.368,6.203,148.636
C06200=1192.000,140.578,-53.540,-178.371,6.202,148.637
C06201=1192.004,140.329,-53.520,-178.373,6.200,148.637
C06202=1192.009,140.080,-53.499,-178.376,6.199,148.638
C06203=1192.014,139.831,-53.478,-178.379,6.197,148.638
C06204=1192.019,139.582,-53.458,-178.381,6.196,148.639
C06205=1192.023,139.333,-53.438,-178.384,6.194,148.639
C06206=1192.028,139.083,-53.417,-178.387,6.193,148.639
C06207=1192.033,138.834,-53.397,-178.389,6.192,148.640
C06208=1192.038,138.586,-53.377,-178.392,6.190,148.640
C06209=1192.043,138.336,-53.356,-178.395,6.189,148.641
C06210=1192.048,138.087,-53.336,-178.397,6.187,148.641
C06211=1192.052,137.838,-53.315,-178.399,6.186,148.642
C06212=1192.057,137.589,-53.295,-178.403,6.184,148.642
C06213=1192.062,137.340,-53.275,-178.405,6.183,148.643
C06214=1192.066,137.091,-53.254,-178.407,6.182,148.643
C06215=1192.071,136.841,-53.233,-178.410,6.180,148.643
C06216=1192.076,136.592,-53.213,-178.413,6.179,148.644
C06217=1192.081,136.343,-53.193,-178.415,6.178,148.644
C06218=1192.085,136.094,-53.173,-178.418,6.176,148.645
C06219=1192.090,135.845,-53.152,-178.421,6.174,148.645
C06220=1192.095,135.596,-53.132,-178.424,6.173,148.646
C06221=1192.099,135.346,-53.112,-178.426,6.172,148.646
C06222=1192.104,135.098,-53.092,-178.429,6.170,148.647
C06223=1192.110,134.849,-53.071,-178.431,6.168,148.647
C06224=1192.114,134.599,-53.051,-178.434,6.168,148.648
C06225=1192.119,134.350,-53.031,-178.437,6.166,148.648
C06226=1192.123,134.101,-53.011,-178.439,6.164,148.648
C06227=1192.128,133.852,-52.991,-178.442,6.163,148.649
C06228=1192.133,133.602,-52.970,-178.445,6.162,148.649
C06229=1192.138,133.353,-52.950,-178.447,6.160,148.650
C06230=1192.143,133.085,-52.928,-178.450,6.159,148.650
C06231=1192.148,132.816,-52.907,-178.453,6.158,148.651
C06232=1192.153,132.548,-52.885,-178.456,6.156,148.651
C06233=1192.158,132.279,-52.863,-178.459,6.154,148.652
C06234=1192.163,132.030,-52.843,-178.461,6.153,148.652
C06235=1192.168,131.780,-52.823,-178.464,6.152,148.653
C06236=1192.173,131.532,-52.803,-178.466,6.150,148.653
C06237=1192.177,131.283,-52.783,-178.469,6.149,148.654
C06238=1192.183,131.033,-52.763,-178.471,6.148,148.654
C06239=1192.187,130.784,-52.742,-178.474,6.146,148.655
C06240=1192.192,130.535,-52.723,-178.477,6.144,148.655
C06241=1192.196,130.286,-52.702,-178.479,6.143,148.655
C06242=1192.202,130.037,-52.683,-178.482,6.142,148.656
C06243=1192.206,129.788,-52.663,-178.485,6.140,148.656
C06244=1192.211,129.538,-52.643,-178.487,6.139,148.657
C06245=1192.215,129.289,-52.623,-178.490,6.138,148.657
C06246=1192.221,129.040,-52.603,-178.493,6.136,148.658
C06247=1192.225,128.791,-52.584,-178.495,6.135,148.658
C06248=1192.230,128.542,-52.563,-178.498,6.133,148.659
C06249=1192.234,128.292,-52.544,-178.501,6.133,148.659
C06250=1192.239,128.043,-52.523,-178.503,6.131,148.660
C06251=1192.244,127.795,-52.504,-178.506,6.129,148.660
C06252=1192.249,127.546,-52.484,-178.509,6.129,148.661
C06253=1192.253,127.296,-52.464,-178.511,6.127,148.661
C06254=1192.258,127.047,-52.444,-178.514,6.125,148.661
C06255=1192.263,126.798,-52.424,-178.517,6.125,148.662
C06256=1192.268,126.549,-52.405,-178.519,6.123,148.662
C06257=1192.273,126.299,-52.385,-178.522,6.121,148.663
C06258=1192.277,126.050,-52.365,-178.525,6.121,148.663
C06259=1192.282,125.801,-52.345,-178.527,6.119,148.664
C06260=1192.287,125.552,-52.326,-178.529,6.118,148.664
C06261=1192.292,125.303,-52.305,-178.533,6.116,148.665
C06262=1192.296,125.053,-52.286,-178.535,6.115,148.665
C06263=1192.302,124.804,-52.266,-178.537,6.114,148.666
C06264=1192.306,124.555,-52.246,-178.541,6.112,148.666
C06265=1192.311,124.306,-52.226,-178.543,6.111,148.667
C06266=1192.316,124.057,-52.207,-178.545,6.110,148.667
C06267=1192.321,123.807,-52.187,-178.549,6.108,148.668
C06268=1192.325,123.558,-52.167,-178.551,6.107,148.668
C06269=1192.330,123.309,-52.147,-178.553,6.106,148.669
C06270=1192.336,123.060,-52.128,-178.556,6.105,148.669
C06271=1192.340,122.811,-52.109,-178.559,6.103,148.670
C06272=1192.344,122.561,-52.089,-178.561,6.101,148.670
C06273=1192.349,122.313,-52.069,-178.564,6.101,148.671
C06274=1192.354,122.063,-52.050,-178.567,6.099,148.671
C06275=1192.359,121.814,-52.030,-178.569,6.098,148.671
C06276=1192.364,121.565,-52.011,-178.572,6.097,148.672
C06277=1192.369,121.315,-51.991,-178.575,6.095,148.672
C06278=1192.373,121.066,-51.972,-178.577,6.094,148.673
C06279=1192.378,120.817,-51.953,-178.580,6.093,148.673
C06280=1192.383,120.568,-51.932,-178.582,6.092,148.674
C06281=1192.387,120.319,-51.913,-178.585,6.090,148.674
C06282=1192.393,120.070,-51.893,-178.588,6.089,148.675
C06283=1192.397,119.820,-51.874,-178.590,6.088,148.675
C06284=1192.402,119.572,-51.855,-178.593,6.086,148.676
C06285=1192.407,119.322,-51.835,-178.595,6.085,148.676
C06286=1192.412,119.073,-51.816,-178.598,6.084,148.677
C06287=1192.417,118.824,-51.796,-178.601,6.083,148.677
C06288=1192.421,118.574,-51.777,-178.603,6.081,148.678
C06289=1192.426,118.326,-51.758,-178.606,6.079,148.678
C06290=1192.431,118.076,-51.738,-178.609,6.079,148.679
C06291=1192.436,117.826,-51.719,-178.611,6.077,148.679
C06292=1192.440,117.578,-51.700,-178.614,6.076,148.680
C06293=1192.445,117.328,-51.680,-178.617,6.075,148.680
C06294=1192.450,117.079,-51.661,-178.619,6.074,148.681
C06295=1192.455,116.830,-51.641,-178.622,6.072,148.681
C06296=1192.459,116.581,-51.622,-178.625,6.071,148.682
C06297=1192.465,116.332,-51.603,-178.627,6.070,148.682
C06298=1192.469,116.082,-51.583,-178.630,6.068,148.683
C06299=1192.475,115.833,-51.564,-178.632,6.067,148.683
C06300=1192.479,115.584,-51.545,-178.635,6.066,148.684
C06301=1192.484,115.335,-51.526,-178.638,6.065,148.684
C06302=1192.489,115.086,-51.506,-178.640,6.063,148.685
C06303=1192.494,114.836,-51.488,-178.643,6.063,148.685
C06304=1192.498,114.587,-51.468,-178.646,6.061,148.686
C06305=1192.504,114.338,-51.449,-178.648,6.059,148.686
C06306=1192.508,114.089,-51.430,-178.651,6.059,148.687
C06307=1192.512,113.839,-51.410,-178.654,6.057,148.687
C06308=1192.518,113.590,-51.391,-178.656,6.056,148.688
C06309=1192.522,113.341,-51.372,-178.659,6.055,148.688
C06310=1192.527,113.092,-51.354,-178.661,6.054,148.688
C06311=1192.531,112.842,-51.334,-178.664,6.052,148.689
C06312=1192.537,112.593,-51.315,-178.666,6.051,148.690
C06313=1192.542,112.344,-51.296,-178.669,6.050,148.690
C06314=1192.546,112.095,-51.277,-178.672,6.049,148.691
C06315=1192.551,111.845,-51.258,-178.674,6.047,148.691
C06316=1192.556,111.597,-51.239,-178.677,6.047,148.692
C06317=1192.561,111.347,-51.220,-178.680,6.045,148.692
C06318=1192.566,111.098,-51.200,-178.683,6.044,148.693
C06319=1192.571,110.849,-51.182,-178.685,6.043,148.693
C06320=1192.576,110.599,-51.163,-178.688,6.041,148.693
C06321=1192.580,110.351,-51.144,-178.690,6.040,148.694
C06322=1192.585,110.101,-51.125,-178.693,6.039,148.694
C06323=1192.590,109.852,-51.106,-178.696,6.038,148.695
C06324=1192.595,109.603,-51.087,-178.698,6.036,148.696
C06325=1192.599,109.353,-51.069,-178.701,6.036,148.696
C06326=1192.604,109.104,-51.049,-178.704,6.034,148.697
C06327=1192.609,108.855,-51.030,-178.706,6.033,148.697
C06328=1192.614,108.605,-51.011,-178.709,6.032,148.698
C06329=1192.618,108.357,-50.993,-178.711,6.031,148.698
C06330=1192.624,108.108,-50.973,-178.714,6.029,148.699
C06331=1192.628,107.858,-50.955,-178.716,6.028,148.699
C06332=1192.633,107.609,-50.936,-178.720,6.027,148.700
C06333=1192.638,107.359,-50.917,-178.722,6.026,148.700
C06334=1192.643,107.091,-50.897,-178.725,6.025,148.701
C06335=1192.649,106.823,-50.877,-178.728,6.023,148.701
C06336=1192.653,106.554,-50.856,-178.730,6.022,148.702
C06337=1192.659,106.286,-50.836,-178.733,6.021,148.702
C06338=1192.664,106.037,-50.817,-178.736,6.019,148.703
C06339=1192.669,105.787,-50.799,-178.738,6.018,148.703
C06340=1192.673,105.538,-50.780,-178.741,6.018,148.704
C06341=1192.678,105.288,-50.762,-178.744,6.016,148.704
C06342=1192.683,105.040,-50.742,-178.746,6.015,148.705
C06343=1192.688,104.790,-50.724,-178.749,6.014,148.705
C06344=1192.693,104.541,-50.705,-178.751,6.013,148.706
C06345=1192.698,104.292,-50.687,-178.754,6.011,148.706
C06346=1192.702,104.043,-50.668,-178.756,6.010,148.707
C06347=1192.707,103.793,-50.649,-178.759,6.009,148.707
C06348=1192.712,103.544,-50.630,-178.762,6.008,148.708
C06349=1192.718,103.295,-50.612,-178.765,6.007,148.709
C06350=1192.722,103.046,-50.593,-178.767,6.006,148.709
C06351=1192.726,102.796,-50.575,-178.770,6.004,148.710
C06352=1192.732,102.547,-50.556,-178.772,6.003,148.710
C06353=1192.736,102.298,-50.537,-178.775,6.002,148.711
C06354=1192.741,102.049,-50.519,-178.778,6.001,148.711
C06355=1192.746,101.800,-50.500,-178.780,5.999,148.711
C06356=1192.751,101.550,-50.481,-178.783,5.999,148.712
C06357=1192.756,101.301,-50.463,-178.786,5.997,148.713
C06358=1192.760,101.052,-50.445,-178.788,5.997,148.713
C06359=1192.765,100.802,-50.426,-178.791,5.995,148.714
C06360=1192.770,100.553,-50.408,-178.794,5.994,148.714
C06361=1192.775,100.304,-50.389,-178.796,5.993,148.715
C06362=1192.780,100.055,-50.371,-178.799,5.992,148.715
C06363=1192.785,99.805,-50.352,-178.801,5.991,148.716
C06364=1192.789,99.556,-50.333,-178.804,5.990,148.716
C06365=1192.794,99.307,-50.316,-178.806,5.989,148.717
C06366=1192.799,99.057,-50.297,-178.810,5.987,148.717
C06367=1192.804,98.808,-50.279,-178.812,5.986,148.718
C06368=1192.809,98.559,-50.260,-178.814,5.985,148.718
C06369=1192.814,98.310,-50.242,-178.817,5.984,148.719
C06370=1192.819,98.060,-50.223,-178.820,5.982,148.719
C06371=1192.824,97.811,-50.205,-178.822,5.982,148.720
C06372=1192.829,97.561,-50.187,-178.824,5.981,148.720
C06373=1192.833,97.313,-50.168,-178.828,5.979,148.721
C06374=1192.837,97.063,-50.150,-178.830,5.979,148.721
C06375=1192.843,96.813,-50.131,-178.833,5.977,148.722
C06376=1192.848,96.564,-50.113,-178.835,5.976,148.722
C06377=1192.853,96.315,-50.095,-178.838,5.975,148.723
C06378=1192.858,96.067,-50.077,-178.840,5.974,148.724
C06379=1192.862,95.817,-50.058,-178.843,5.973,148.724
C06380=1192.867,95.568,-50.040,-178.846,5.972,148.725
C06381=1192.872,95.318,-50.022,-178.848,5.971,148.725
C06382=1192.877,95.069,-50.004,-178.851,5.969,148.726
C06383=1192.882,94.820,-49.986,-178.854,5.969,148.726
C06384=1192.887,94.570,-49.968,-178.856,5.967,148.727
C06385=1192.891,94.321,-49.950,-178.859,5.966,148.727
C06386=1192.896,94.071,-49.932,-178.861,5.966,148.728
C06387=1192.901,93.822,-49.914,-178.864,5.964,148.728
C06388=1192.906,93.574,-49.895,-178.867,5.963,148.729
C06389=1192.910,93.324,-49.877,-178.870,5.962,148.729
C06390=1192.916,93.074,-49.858,-178.872,5.961,148.730
C06391=1192.921,92.825,-49.840,-178.874,5.960,148.731
C06392=1192.926,92.576,-49.822,-178.877,5.959,148.731
C06393=1192.931,92.327,-49.804,-178.880,5.958,148.732
C06394=1192.936,92.078,-49.786,-178.882,5.956,148.732
C06395=1192.940,91.828,-49.768,-178.885,5.956,148.733
C06396=1192.945,91.579,-49.750,-178.888,5.954,148.733
C06397=1192.950,91.329,-49.732,-178.890,5.954,148.734
C06398=1192.955,91.080,-49.714,-178.893,5.953,148.734
C06399=1192.959,90.831,-49.696,-178.896,5.951,148.735
C06400=1192.964,90.582,-49.678,-178.898,5.950,148.735
C06401=1192.970,90.332,-49.661,-178.901,5.949,148.736
C06402=1192.975,90.083,-49.643,-178.903,5.948,148.736
C06403=1192.979,89.833,-49.624,-178.906,5.947,148.737
C06404=1192.984,89.584,-49.606,-178.909,5.946,148.737
C06405=1192.989,89.335,-49.588,-178.911,5.945,148.738
C06406=1192.994,89.086,-49.570,-178.914,5.943,148.738
C06407=1192.998,88.836,-49.552,-178.917,5.943,148.739
C06408=1193.003,88.587,-49.534,-178.919,5.942,148.739
C06409=1193.008,88.338,-49.516,-178.922,5.941,148.740
C06410=1193.014,88.088,-49.499,-178.924,5.940,148.741
C06411=1193.018,87.839,-49.481,-178.927,5.939,148.741
C06412=1193.023,87.590,-49.463,-178.930,5.938,148.742
C06413=1193.028,87.341,-49.445,-178.932,5.937,148.742
C06414=1193.033,87.092,-49.427,-178.935,5.935,148.743
C06415=1193.037,86.842,-49.409,-178.937,5.935,148.743
C06416=1193.042,86.592,-49.392,-178.940,5.934,148.744
C06417=1193.047,86.343,-49.374,-178.943,5.932,148.744
C06418=1193.052,86.094,-49.356,-178.945,5.932,148.745
C06419=1193.057,85.845,-49.338,-178.947,5.931,148.745
C06420=1193.062,85.595,-49.321,-178.951,5.929,148.746
C06421=1193.067,85.346,-49.303,-178.953,5.928,148.747
C06422=1193.072,85.096,-49.285,-178.956,5.927,148.747
C06423=1193.077,84.847,-49.267,-178.958,5.926,148.748
C06424=1193.082,84.597,-49.250,-178.961,5.926,148.748
C06425=1193.086,84.349,-49.232,-178.963,5.924,148.749
C06426=1193.091,84.099,-49.214,-178.966,5.923,148.749
C06427=1193.096,83.850,-49.197,-178.969,5.923,148.750
C06428=1193.101,83.600,-49.179,-178.971,5.921,148.750
C06429=1193.106,83.351,-49.161,-178.974,5.921,148.751
C06430=1193.111,83.102,-49.144,-178.976,5.920,148.752
C06431=1193.115,82.853,-49.127,-178.979,5.918,148.752
C06432=1193.120,82.603,-49.109,-178.981,5.917,148.753
C06433=1193.126,82.354,-49.091,-178.984,5.917,148.753
C06434=1193.130,82.104,-49.073,-178.987,5.915,148.754
C06435=1193.135,81.855,-49.055,-178.989,5.915,148.754
C06436=1193.140,81.606,-49.039,-178.992,5.914,148.755
C06437=1193.145,81.357,-49.021,-178.995,5.912,148.755
C06438=1193.150,81.088,-49.002,-178.997,5.912,148.756
C06439=1193.156,80.820,-48.983,-179.001,5.910,148.757
C06440=1193.161,80.551,-48.964,-179.003,5.909,148.757
C06441=1193.166,80.283,-48.945,-179.006,5.908,148.758
C06442=1193.171,80.034,-48.928,-179.009,5.907,148.758
C06443=1193.176,79.784,-48.910,-179.011,5.906,148.759
C06444=1193.181,79.535,-48.893,-179.014,5.905,148.759
C06445=1193.186,79.285,-48.875,-179.016,5.904,148.760
C06446=1193.190,79.036,-48.858,-179.019,5.903,148.761
C06447=1193.195,78.787,-48.840,-179.021,5.902,148.761
C06448=1193.201,78.538,-48.823,-179.024,5.901,148.762
C06449=1193.205,78.289,-48.806,-179.027,5.900,148.762
C06450=1193.210,78.039,-48.789,-179.029,5.899,148.763
C06451=1193.215,77.790,-48.771,-179.032,5.899,148.763
C06452=1193.220,77.540,-48.754,-179.035,5.897,148.764
C06453=1193.225,77.291,-48.736,-179.037,5.896,148.764
C06454=1193.230,77.041,-48.719,-179.040,5.895,148.765
C06455=1193.234,76.792,-48.702,-179.042,5.895,148.766
C06456=1193.239,76.543,-48.684,-179.045,5.894,148.766
C06457=1193.245,76.293,-48.667,-179.047,5.893,148.767
C06458=1193.249,76.045,-48.650,-179.050,5.892,148.767
C06459=1193.255,75.795,-48.633,-179.053,5.890,148.768
C06460=1193.260,75.545,-48.615,-179.055,5.890,148.768
C06461=1193.264,75.296,-48.598,-179.058,5.889,148.769
C06462=1193.269,75.047,-48.581,-179.061,5.888,148.769
C06463=1193.274,74.797,-48.563,-179.063,5.887,148.770
C06464=1193.279,74.548,-48.546,-179.066,5.886,148.771
C06465=1193.284,74.299,-48.529,-179.069,5.885,148.771
C06466=1193.289,74.050,-48.512,-179.071,5.884,148.772
C06467=1193.294,73.800,-48.495,-179.074,5.883,148.772
C06468=1193.298,73.551,-48.478,-179.076,5.883,148.773
C06469=1193.303,73.301,-48.461,-179.079,5.881,148.773
C06470=1193.308,73.052,-48.443,-179.082,5.880,148.774
C06471=1193.313,72.802,-48.426,-179.084,5.880,148.774
C06472=1193.319,72.553,-48.409,-179.087,5.878,148.775
C06473=1193.323,72.304,-48.392,-179.090,5.878,148.776
C06474=1193.328,72.054,-48.374,-179.092,5.877,148.776
C06475=1193.333,71.805,-48.358,-179.094,5.876,148.777
C06476=1193.338,71.555,-48.340,-179.097,5.874,148.777
C06477=1193.343,71.306,-48.324,-179.100,5.874,148.778
C06478=1193.348,71.057,-48.306,-179.102,5.873,148.778
C06479=1193.352,70.808,-48.290,-179.105,5.872,148.779
C06480=1193.357,70.558,-48.272,-179.108,5.871,148.780
C06481=1193.362,70.308,-48.256,-179.110,5.870,148.780
C06482=1193.368,70.059,-48.239,-179.112,5.870,148.781
C06483=1193.372,69.811,-48.221,-179.115,5.868,148.781
C06484=1193.377,69.561,-48.204,-179.118,5.867,148.782
C06485=1193.382,69.311,-48.187,-179.120,5.867,148.783
C06486=1193.387,69.062,-48.170,-179.123,5.865,148.783
C06487=1193.392,68.813,-48.154,-179.126,5.865,148.784
C06488=1193.397,68.563,-48.137,-179.128,5.864,148.784
C06489=1193.402,68.313,-48.120,-179.130,5.863,148.785
C06490=1193.407,68.065,-48.102,-179.134,5.862,148.785
C06491=1193.412,67.815,-48.086,-179.136,5.861,148.786
C06492=1193.416,67.566,-48.069,-179.138,5.860,148.786
C06493=1193.421,67.316,-48.052,-179.141,5.860,148.787
C06494=1193.426,67.067,-48.035,-179.144,5.858,148.788
C06495=1193.432,66.818,-48.018,-179.146,5.858,148.788
C06496=1193.436,66.568,-48.001,-179.149,5.857,148.789
C06497=1193.441,66.319,-47.985,-179.151,5.856,148.789
C06498=1193.446,66.069,-47.968,-179.154,5.855,148.790
C06499=1193.451,65.820,-47.951,-179.157,5.854,148.790
C06500=1193.456,65.570,-47.934,-179.159,5.853,148.791
C06501=1193.461,65.321,-47.918,-179.162,5.853,148.792
C06502=1193.466,65.072,-47.901,-179.165,5.851,148.792
C06503=1193.471,64.822,-47.884,-179.167,5.851,148.793
C06504=1193.476,64.573,-47.867,-179.169,5.850,148.793
C06505=1193.480,64.324,-47.851,-179.172,5.849,148.794
C06506=1193.486,64.074,-47.833,-179.175,5.848,148.795
C06507=1193.490,63.825,-47.817,-179.177,5.847,148.795
C06508=1193.495,63.576,-47.800,-179.180,5.846,148.796
C06509=1193.500,63.326,-47.783,-179.183,5.846,148.796
C06510=1193.505,63.077,-47.767,-179.185,5.844,148.797
C06511=1193.510,62.828,-47.750,-179.188,5.844,148.797
C06512=1193.515,62.578,-47.733,-179.190,5.843,148.798
C06513=1193.520,62.328,-47.717,-179.193,5.842,148.799
C06514=1193.525,62.079,-47.701,-179.196,5.841,148.799
C06515=1193.530,61.830,-47.684,-179.198,5.840,148.800
C06516=1193.535,61.580,-47.667,-179.201,5.839,148.800
C06517=1193.540,61.331,-47.650,-179.203,5.839,148.801
C06518=1193.544,61.082,-47.634,-179.206,5.838,148.801
C06519=1193.549,60.833,-47.617,-179.209,5.837,148.802
C06520=1193.555,60.582,-47.601,-179.211,5.836,148.803
C06521=1193.559,60.333,-47.584,-179.213,5.835,148.803
C06522=1193.564,60.084,-47.568,-179.216,5.835,148.804
C06523=1193.569,59.835,-47.551,-179.219,5.833,148.804
C06524=1193.575,59.585,-47.534,-179.221,5.832,148.805
C06525=1193.580,59.335,-47.518,-179.224,5.832,148.806
C06526=1193.584,59.086,-47.502,-179.226,5.831,148.806
C06527=1193.589,58.837,-47.485,-179.229,5.830,148.807
C06528=1193.594,58.588,-47.469,-179.232,5.829,148.807
C06529=1193.599,58.339,-47.452,-179.234,5.828,148.808
C06530=1193.604,58.088,-47.436,-179.237,5.828,148.808
C06531=1193.609,57.839,-47.419,-179.240,5.827,148.809
C06532=1193.614,57.590,-47.403,-179.242,5.826,148.810
C06533=1193.619,57.340,-47.387,-179.245,5.825,148.810
C06534=1193.624,57.091,-47.370,-179.248,5.824,148.811
C06535=1193.629,56.841,-47.353,-179.250,5.823,148.811
C06536=1193.634,56.593,-47.337,-179.252,5.823,148.812
C06537=1193.639,56.343,-47.321,-179.255,5.822,148.813
C06538=1193.644,56.094,-47.305,-179.258,5.821,148.813
C06539=1193.648,55.844,-47.288,-179.260,5.820,148.814
C06540=1193.653,55.594,-47.272,-179.262,5.819,148.814
C06541=1193.659,55.345,-47.255,-179.265,5.819,148.815
C06542=1193.664,55.077,-47.238,-179.268,5.817,148.816
C06543=1193.669,54.808,-47.220,-179.271,5.817,148.816
C06544=1193.675,54.540,-47.203,-179.274,5.816,148.817
C06545=1193.680,54.272,-47.186,-179.277,5.815,148.818
C06546=1193.685,54.022,-47.170,-179.279,5.814,148.818
C06547=1193.690,53.773,-47.153,-179.282,5.813,148.819
C06548=1193.695,53.523,-47.137,-179.284,5.813,148.819
C06549=1193.700,53.274,-47.120,-179.286,5.812,148.820
C06550=1193.705,53.024,-47.104,-179.290,5.811,148.820
C06551=1193.710,52.775,-47.088,-179.292,5.810,148.821
C06552=1193.715,52.525,-47.072,-179.294,5.809,148.822
C06553=1193.720,52.276,-47.056,-179.297,5.809,148.822
C06554=1193.725,52.026,-47.039,-179.300,5.808,148.823
C06555=1193.730,51.777,-47.024,-179.302,5.807,148.823
C06556=1193.734,51.528,-47.007,-179.305,5.806,148.824
C06557=1193.740,51.278,-46.991,-179.308,5.805,148.825
C06558=1193.744,51.029,-46.975,-179.310,5.805,148.825
C06559=1193.750,50.779,-46.959,-179.312,5.804,148.826
C06560=1193.754,50.530,-46.942,-179.315,5.803,148.826
C06561=1193.760,50.280,-46.927,-179.317,5.803,148.827
C06562=1193.764,50.030,-46.911,-179.320,5.801,148.827
C06563=1193.769,49.781,-46.895,-179.323,5.801,148.828
C06564=1193.774,49.531,-46.879,-179.325,5.800,148.829
C06565=1193.779,49.283,-46.862,-179.328,5.799,148.829
C06566=1193.785,49.033,-46.847,-179.331,5.799,148.830
C06567=1193.789,48.784,-46.830,-179.333,5.798,148.830
C06568=1193.795,48.534,-46.815,-179.336,5.797,148.831
C06569=1193.799,48.284,-46.799,-179.339,5.796,148.832
C06570=1193.804,48.036,-46.783,-179.341,5.795,148.832
C06571=1193.808,47.786,-46.767,-179.343,5.795,148.833
C06572=1193.814,47.537,-46.751,-179.346,5.794,148.834
C06573=1193.819,47.287,-46.735,-179.348,5.793,148.834
C06574=1193.824,47.037,-46.719,-179.351,5.793,148.835
C06575=1193.829,46.789,-46.703,-179.354,5.791,148.835
C06576=1193.834,46.538,-46.687,-179.357,5.791,148.836
C06577=1193.839,46.289,-46.671,-179.359,5.790,148.836
C06578=1193.844,46.040,-46.655,-179.361,5.789,148.837
C06579=1193.849,45.790,-46.639,-179.364,5.789,148.838
C06580=1193.854,45.541,-46.624,-179.366,5.788,148.838
C06581=1193.858,45.291,-46.608,-179.369,5.787,148.839
C06582=1193.863,45.042,-46.592,-179.372,5.786,148.840
C06583=1193.869,44.793,-46.576,-179.374,5.785,148.840
C06584=1193.874,44.543,-46.560,-179.377,5.785,148.841
C06585=1193.879,44.293,-46.545,-179.379,5.784,148.841
C06586=1193.884,44.044,-46.528,-179.382,5.783,148.842
C06587=1193.888,43.795,-46.513,-179.384,5.783,148.842
C06588=1193.893,43.545,-46.497,-179.387,5.782,148.843
C06589=1193.899,43.296,-46.482,-179.390,5.782,148.844
C06590=1193.903,43.046,-46.465,-179.392,5.780,148.844
C06591=1193.909,42.797,-46.449,-179.395,5.780,148.845
C06592=1193.913,42.548,-46.434,-179.398,5.779,148.846
C06593=1193.918,42.298,-46.419,-179.400,5.778,148.846
C06594=1193.924,42.048,-46.403,-179.402,5.778,148.847
C06595=1193.929,41.800,-46.387,-179.405,5.777,148.847
C06596=1193.933,41.550,-46.371,-179.407,5.776,148.848
C06597=1193.938,41.300,-46.356,-179.410,5.776,148.848
C06598=1193.943,41.051,-46.340,-179.413,5.774,148.849
C06599=1193.948,40.801,-46.324,-179.416,5.774,148.850
C06600=1193.954,40.552,-46.309,-179.418,5.773,148.850
C06601=1193.958,40.302,-46.294,-179.420,5.772,148.851
C06602=1193.963,40.052,-46.278,-179.423,5.772,148.852
C06603=1193.968,39.804,-46.261,-179.425,5.771,148.852
C06604=1193.974,39.554,-46.246,-179.428,5.770,148.853
C06605=1193.978,39.305,-46.231,-179.431,5.770,148.853
C06606=1193.983,39.055,-46.215,-179.433,5.769,148.854
C06607=1193.988,38.806,-46.199,-179.435,5.769,148.855
C06608=1193.994,38.556,-46.184,-179.439,5.767,148.855
C06609=1193.998,38.307,-46.169,-179.441,5.767,148.856
C06610=1194.003,38.057,-46.153,-179.443,5.766,148.856
C06611=1194.009,37.808,-46.137,-179.446,5.765,148.857
C06612=1194.013,37.558,-46.122,-179.449,5.765,148.858
C06613=1194.019,37.309,-46.106,-179.451,5.764,148.858
C06614=1194.023,37.059,-46.091,-179.453,5.763,148.859
C06615=1194.028,36.810,-46.076,-179.456,5.763,148.859
C06616=1194.033,36.560,-46.060,-179.459,5.762,148.860
C06617=1194.039,36.311,-46.044,-179.461,5.761,148.861
C06618=1194.043,36.061,-46.029,-179.463,5.761,148.861
C06619=1194.048,35.812,-46.013,-179.467,5.760,148.862
C06620=1194.054,35.562,-45.998,-179.469,5.759,148.862
C06621=1194.058,35.313,-45.983,-179.472,5.758,148.863
C06622=1194.064,35.064,-45.967,-179.474,5.758,148.864
C06623=1194.068,34.814,-45.952,-179.477,5.757,148.864
C06624=1194.073,34.565,-45.936,-179.479,5.756,148.865
C06625=1194.079,34.315,-45.921,-179.482,5.756,148.866
C06626=1194.083,34.066,-45.906,-179.484,5.755,148.866
C06627=1194.089,33.816,-45.891,-179.487,5.755,148.867
C06628=1194.093,33.566,-45.875,-179.489,5.754,148.867
C06629=1194.098,33.317,-45.860,-179.492,5.753,148.868
C06630=1194.104,33.068,-45.844,-179.494,5.753,148.869
C06631=1194.108,32.819,-45.829,-179.497,5.751,148.869
C06632=1194.114,32.569,-45.814,-179.500,5.751,148.870
C06633=1194.118,32.319,-45.799,-179.502,5.750,148.870
C06634=1194.123,32.069,-45.783,-179.505,5.750,148.871
C06635=1194.128,31.820,-45.769,-179.507,5.749,148.872
C06636=1194.133,31.571,-45.753,-179.510,5.748,148.872
C06637=1194.138,31.322,-45.738,-179.512,5.748,148.873
C06638=1194.144,31.072,-45.723,-179.515,5.747,148.874
C06639=1194.148,30.823,-45.708,-179.517,5.746,148.874
C06640=1194.153,30.573,-45.692,-179.520,5.746,148.875
C06641=1194.158,30.323,-45.677,-179.523,5.745,148.875
C06642=1194.163,30.074,-45.662,-179.525,5.744,148.876
C06643=1194.168,29.824,-45.647,-179.527,5.744,148.877
C06644=1194.174,29.575,-45.632,-179.530,5.743,148.877
C06645=1194.178,29.326,-45.617,-179.533,5.743,148.878
C06646=1194.184,29.057,-45.600,-179.536,5.742,148.879
C06647=1194.190,28.788,-45.584,-179.538,5.741,148.879
C06648=1194.195,28.519,-45.568,-179.541,5.741,148.880
C06649=1194.201,28.250,-45.551,-179.543,5.740,148.880
C06650=1194.205,28.001,-45.536,-179.546,5.739,148.881
C06651=1194.210,27.751,-45.522,-179.549,5.739,148.882
C06652=1194.215,27.501,-45.506,-179.551,5.738,148.882
C06653=1194.220,27.252,-45.491,-179.553,5.737,148.883
C06654=1194.225,27.002,-45.476,-179.556,5.737,148.884
C06655=1194.230,26.753,-45.461,-179.559,5.736,148.884
C06656=1194.235,26.504,-45.446,-179.561,5.736,148.885
C06657=1194.240,26.254,-45.431,-179.563,5.735,148.885
C06658=1194.245,26.005,-45.416,-179.567,5.734,148.886
C06659=1194.250,25.756,-45.401,-179.569,5.733,148.887
C06660=1194.255,25.506,-45.387,-179.572,5.733,148.887
C06661=1194.261,25.257,-45.371,-179.574,5.732,148.888
C06662=1194.266,25.007,-45.357,-179.577,5.731,148.889
C06663=1194.270,24.758,-45.342,-179.579,5.731,148.889
C06664=1194.276,24.508,-45.326,-179.582,5.730,148.890
C06665=1194.281,24.259,-45.312,-179.584,5.729,148.890
C06666=1194.285,24.009,-45.296,-179.587,5.729,148.891
C06667=1194.290,23.759,-45.282,-179.590,5.728,148.892
C06668=1194.295,23.510,-45.267,-179.592,5.728,148.892
C06669=1194.300,23.260,-45.252,-179.594,5.727,148.893
C06670=1194.305,23.011,-45.237,-179.597,5.726,148.893
C06671=1194.310,22.761,-45.222,-179.600,5.726,148.894
C06672=1194.315,22.512,-45.207,-179.602,5.725,148.895
C06673=1194.321,22.262,-45.193,-179.604,5.725,148.895
C06674=1194.325,22.013,-45.178,-179.607,5.724,148.896
C06675=1194.330,21.763,-45.163,-179.610,5.724,148.897
C06676=1194.336,21.514,-45.148,-179.612,5.723,148.897
C06677=1194.341,21.264,-45.133,-179.615,5.722,148.898
C06678=1194.345,21.015,-45.118,-179.617,5.722,148.898
C06679=1194.351,20.765,-45.104,-179.620,5.721,148.899
C06680=1194.356,20.516,-45.089,-179.623,5.721,148.900
C06681=1194.361,20.266,-45.074,-179.625,5.720,148.900
C06682=1194.366,20.016,-45.060,-179.627,5.719,148.901
C06683=1194.371,19.767,-45.044,-179.630,5.719,148.902
C06684=1194.376,19.517,-45.030,-179.633,5.718,148.902
C06685=1194.381,19.269,-45.016,-179.635,5.717,148.903
C06686=1194.386,19.019,-45.001,-179.637,5.717,148.903
C06687=1194.392,18.769,-44.986,-179.640,5.716,148.904
C06688=1194.396,18.520,-44.971,-179.643,5.716,148.905
C06689=1194.401,18.270,-44.957,-179.645,5.715,148.905
C06690=1194.406,18.020,-44.943,-179.648,5.715,148.906
C06691=1194.411,17.771,-44.928,-179.650,5.714,148.907
C06692=1194.417,17.521,-44.913,-179.653,5.714,148.907
C06693=1194.422,17.272,-44.899,-179.655,5.713,148.908
C06694=1194.426,17.023,-44.884,-179.658,5.712,148.908
C06695=1194.431,16.773,-44.869,-179.660,5.712,148.909
C06696=1194.436,16.523,-44.855,-179.663,5.711,148.910
C06697=1194.442,16.274,-44.840,-179.666,5.711,148.911
C06698=1194.447,16.024,-44.825,-179.668,5.710,148.911
C06699=1194.452,15.774,-44.811,-179.670,5.709,148.912
C06700=1194.456,15.525,-44.796,-179.673,5.709,148.912
C06701=1194.462,15.276,-44.782,-179.676,5.708,148.913
C06702=1194.467,15.027,-44.768,-179.678,5.707,148.913
C06703=1194.472,14.777,-44.754,-179.680,5.707,148.914
C06704=1194.477,14.527,-44.738,-179.683,5.706,148.915
C06705=1194.482,14.278,-44.724,-179.686,5.706,148.916
C06706=1194.487,14.028,-44.709,-179.688,5.705,148.916
C06707=1194.492,13.778,-44.695,-179.691,5.705,148.917
C06708=1194.497,13.529,-44.681,-179.693,5.704,148.917
C06709=1194.501,13.279,-44.666,-179.696,5.704,148.918
C06710=1194.507,13.030,-44.652,-179.699,5.703,148.919
C06711=1194.512,12.781,-44.638,-179.700,5.703,148.919
C06712=1194.517,12.531,-44.623,-179.703,5.703,148.920
C06713=1194.523,12.281,-44.609,-179.705,5.702,148.921
C06714=1194.528,12.031,-44.594,-179.708,5.702,148.921
C06715=1194.532,11.782,-44.579,-179.710,5.701,148.922
C06716=1194.538,11.533,-44.565,-179.713,5.700,148.922
C06717=1194.543,11.284,-44.551,-179.716,5.700,148.923
C06718=1194.548,11.034,-44.537,-179.718,5.699,148.924
C06719=1194.553,10.784,-44.523,-179.720,5.698,148.924
C06720=1194.558,10.534,-44.508,-179.723,5.698,148.925
C06721=1194.563,10.285,-44.494,-179.726,5.697,148.926
C06722=1194.568,10.036,-44.480,-179.728,5.697,148.926
C06723=1194.573,9.786,-44.466,-179.731,5.696,148.927
C06724=1194.578,9.537,-44.451,-179.733,5.695,148.927
C06725=1194.583,9.287,-44.437,-179.736,5.695,148.928
C06726=1194.588,9.037,-44.422,-179.738,5.694,148.929
C06727=1194.593,8.788,-44.408,-179.741,5.694,148.929
C06728=1194.598,8.539,-44.394,-179.743,5.693,148.930
C06729=1194.603,8.289,-44.380,-179.746,5.693,148.931
C06730=1194.608,8.039,-44.365,-179.749,5.692,148.931
C06731=1194.613,7.790,-44.351,-179.751,5.692,148.932
C06732=1194.619,7.541,-44.337,-179.754,5.691,148.933
C06733=1194.624,7.291,-44.323,-179.755,5.691,148.933
C06734=1194.628,7.041,-44.309,-179.758,5.691,148.934
C06735=1194.633,6.791,-44.294,-179.761,5.690,148.934
C06736=1194.638,6.542,-44.280,-179.763,5.690,148.935
C06737=1194.644,6.293,-44.266,-179.766,5.689,148.936
C06738=1194.649,6.043,-44.252,-179.768,5.688,148.936
C06739=1194.654,5.793,-44.238,-179.771,5.688,148.937
C06740=1194.658,5.544,-44.224,-179.774,5.687,148.938
C06741=1194.664,5.295,-44.210,-179.776,5.687,148.938
C06742=1194.669,5.045,-44.197,-179.778,5.686,148.939
C06743=1194.674,4.795,-44.182,-179.781,5.685,148.940
C06744=1194.679,4.545,-44.168,-179.784,5.685,148.940
C06745=1194.684,4.296,-44.154,-179.786,5.684,148.941
C06746=1194.689,4.046,-44.140,-179.789,5.684,148.942
C06747=1194.694,3.797,-44.126,-179.791,5.684,148.942
C06748=1194.699,3.547,-44.111,-179.793,5.683,148.943
C06749=1194.705,3.298,-44.097,-179.796,5.683,148.943
C06750=1194.710,3.029,-44.082,-179.798,5.682,148.944
C06751=1194.715,2.759,-44.068,-179.801,5.682,148.945
C06752=1194.720,2.490,-44.053,-179.804,5.681,148.945
C06753=1194.726,2.222,-44.038,-179.807,5.680,148.946
C06754=1194.731,1.972,-44.024,-179.810,5.680,148.947
C06755=1194.736,1.722,-44.010,-179.811,5.680,148.947
C06756=1194.741,1.472,-43.996,-179.814,5.679,148.948
C06757=1194.747,1.223,-43.982,-179.817,5.679,148.949
C06758=1194.752,0.973,-43.967,-179.819,5.678,148.949
C06759=1194.756,0.723,-43.954,-179.822,5.678,148.950
C06760=1194.762,0.474,-43.940,-179.824,5.677,148.951
C06761=1194.767,0.225,-43.926,-179.827,5.676,148.951
C06762=1194.772,-0.025,-43.912,-179.829,5.676,148.952
C06763=1194.778,-0.275,-43.899,-179.832,5.675,148.953
C06764=1194.782,-0.524,-43.885,-179.835,5.675,148.953
C06765=1194.787,-0.774,-43.871,-179.836,5.675,148.954
C06766=1194.792,-1.023,-43.857,-179.839,5.674,148.954
C06767=1194.798,-1.273,-43.843,-179.842,5.674,148.955
C06768=1194.803,-1.523,-43.829,-179.844,5.673,148.956
C06769=1194.807,-1.771,-43.816,-179.847,5.673,148.957
C06770=1194.813,-2.022,-43.802,-179.849,5.672,148.957
C06771=1194.818,-2.271,-43.788,-179.852,5.672,148.958
C06772=1194.822,-2.520,-43.775,-179.854,5.671,148.958
C06773=1194.827,-2.770,-43.760,-179.857,5.671,148.959
C06774=1194.833,-3.020,-43.747,-179.859,5.670,148.959
C06775=1194.838,-3.269,-43.733,-179.861,5.670,148.960
C06776=1194.842,-3.519,-43.719,-179.864,5.670,148.961
C06777=1194.848,-3.768,-43.706,-179.867,5.669,148.962
C06778=1194.853,-4.018,-43.692,-179.869,5.669,148.962
C06779=1194.859,-4.268,-43.678,-179.871,5.668,148.963
C06780=1194.863,-4.517,-43.665,-179.874,5.667,148.963
C06781=1194.868,-4.767,-43.650,-179.877,5.667,148.964
C06782=1194.874,-5.016,-43.637,-179.879,5.666,148.965
C06783=1194.878,-5.266,-43.624,-179.882,5.666,148.965
C06784=1194.884,-5.515,-43.610,-179.884,5.666,148.966
C06785=1194.889,-5.765,-43.596,-179.886,5.665,148.967
C06786=1194.893,-6.014,-43.582,-179.889,5.665,148.967
C06787=1194.899,-6.264,-43.569,-179.892,5.664,148.968
C06788=1194.904,-6.514,-43.555,-179.894,5.664,148.969
C06789=1194.909,-6.763,-43.542,-179.896,5.663,148.969
C06790=1194.914,-7.013,-43.528,-179.899,5.663,148.970
C06791=1194.919,-7.262,-43.515,-179.902,5.662,148.971
C06792=1194.924,-7.512,-43.501,-179.904,5.662,148.971
C06793=1194.930,-7.762,-43.488,-179.906,5.662,148.972
C06794=1194.934,-8.011,-43.474,-179.909,5.661,148.972
C06795=1194.940,-8.261,-43.461,-179.911,5.661,148.973
C06796=1194.944,-8.510,-43.447,-179.914,5.660,148.974
C06797=1194.950,-8.760,-43.434,-179.917,5.660,148.974
C06798=1194.955,-9.009,-43.420,-179.919,5.659,148.975
C06799=1194.960,-9.259,-43.407,-179.921,5.659,148.976
C06800=1194.965,-9.508,-43.393,-179.923,5.659,148.976
C06801=1194.970,-9.758,-43.380,-179.926,5.658,148.977
C06802=1194.975,-10.007,-43.366,-179.929,5.658,148.978
C06803=1194.981,-10.258,-43.353,-179.931,5.657,148.978
C06804=1194.986,-10.507,-43.340,-179.934,5.656,148.979
C06805=1194.991,-10.757,-43.326,-179.936,5.656,148.980
C06806=1194.996,-11.006,-43.313,-179.938,5.656,148.980
C06807=1195.001,-11.256,-43.299,-179.941,5.656,148.981
C06808=1195.006,-11.505,-43.286,-179.944,5.655,148.982
C06809=1195.011,-11.755,-43.273,-179.946,5.654,148.982
C06810=1195.016,-12.004,-43.259,-179.948,5.654,148.983
C06811=1195.021,-12.254,-43.246,-179.951,5.653,148.983
C06812=1195.026,-12.503,-43.233,-179.954,5.653,148.984
C06813=1195.031,-12.753,-43.219,-179.956,5.653,148.985
C06814=1195.037,-13.003,-43.206,-179.958,5.652,148.985
C06815=1195.041,-13.252,-43.192,-179.961,5.652,148.986
C06816=1195.047,-13.502,-43.179,-179.963,5.651,148.987
C06817=1195.052,-13.752,-43.166,-179.966,5.651,148.987
C06818=1195.057,-14.001,-43.153,-179.969,5.651,148.988
C06819=1195.062,-14.251,-43.139,-179.970,5.650,148.989
C06820=1195.067,-14.500,-43.126,-179.973,5.650,148.989
C06821=1195.072,-14.751,-43.113,-179.976,5.650,148.990
C06822=1195.077,-14.999,-43.100,-179.978,5.649,148.991
C06823=1195.083,-15.249,-43.086,-179.981,5.649,148.991
C06824=1195.088,-15.499,-43.073,-179.983,5.648,148.992
C06825=1195.092,-15.748,-43.060,-179.985,5.648,148.992
C06826=1195.098,-15.998,-43.047,-179.988,5.648,148.993
C06827=1195.103,-16.247,-43.034,-179.990,5.647,148.994
C06828=1195.108,-16.498,-43.020,-179.993,5.647,148.995
C06829=1195.113,-16.747,-43.008,-179.995,5.646,148.995
C06830=1195.119,-16.996,-42.994,-179.998,5.645,148.996
C06831=1195.123,-17.246,-42.981,-180.000,5.646,148.996
C06832=1195.128,-17.495,-42.968,179.997,5.645,148.997
C06833=1195.134,-17.746,-42.955,179.995,5.645,148.998
C06834=1195.138,-17.994,-42.941,179.993,5.644,148.998
C06835=1195.144,-18.244,-42.928,179.990,5.643,148.999
C06836=1195.149,-18.494,-42.915,179.987,5.643,149.000
C06837=1195.154,-18.743,-42.903,179.985,5.643,149.000
C06838=1195.159,-18.994,-42.889,179.983,5.643,149.001
C06839=1195.164,-19.243,-42.876,179.980,5.642,149.002
C06840=1195.169,-19.492,-42.864,179.978,5.641,149.002
C06841=1195.174,-19.742,-42.850,179.975,5.641,149.003
C06842=1195.180,-19.991,-42.837,179.973,5.641,149.004
C06843=1195.185,-20.241,-42.824,179.970,5.641,149.004
C06844=1195.190,-20.491,-42.811,179.968,5.640,149.005
C06845=1195.195,-20.740,-42.798,179.965,5.640,149.005
C06846=1195.201,-20.990,-42.785,179.963,5.639,149.006
C06847=1195.205,-21.240,-42.772,179.960,5.639,149.007
C06848=1195.211,-21.489,-42.759,179.958,5.639,149.008
C06849=1195.216,-21.740,-42.746,179.956,5.638,149.008
C06850=1195.221,-21.989,-42.733,179.953,5.638,149.009
C06851=1195.226,-22.238,-42.720,179.951,5.637,149.009
C06852=1195.230,-22.488,-42.707,179.948,5.637,149.010
C06853=1195.236,-22.737,-42.694,179.946,5.637,149.011
C06854=1195.241,-23.007,-42.680,179.943,5.637,149.011
C06855=1195.247,-23.276,-42.666,179.941,5.636,149.012
C06856=1195.252,-23.546,-42.653,179.938,5.636,149.013
C06857=1195.258,-23.816,-42.638,179.935,5.635,149.014
C06858=1195.263,-24.066,-42.626,179.933,5.635,149.014
C06859=1195.268,-24.315,-42.613,179.930,5.634,149.015
C06860=1195.273,-24.565,-42.600,179.928,5.633,149.015
C06861=1195.279,-24.814,-42.587,179.926,5.634,149.016
C06862=1195.284,-25.064,-42.574,179.923,5.633,149.017
C06863=1195.289,-25.313,-42.562,179.920,5.633,149.018
C06864=1195.294,-25.563,-42.549,179.918,5.632,149.018
C06865=1195.299,-25.813,-42.536,179.915,5.632,149.019
C06866=1195.305,-26.062,-42.523,179.913,5.632,149.019
C06867=1195.309,-26.312,-42.510,179.911,5.631,149.020
C06868=1195.314,-26.561,-42.497,179.908,5.631,149.021
C06869=1195.320,-26.811,-42.486,179.906,5.630,149.021
C06870=1195.326,-27.061,-42.472,179.904,5.630,149.022
C06871=1195.330,-27.311,-42.459,179.901,5.630,149.023
C06872=1195.335,-27.560,-42.447,179.898,5.630,149.023
C06873=1195.340,-27.810,-42.434,179.896,5.629,149.024
C06874=1195.345,-28.059,-42.422,179.893,5.629,149.025
C06875=1195.350,-28.309,-42.409,179.892,5.629,149.025
C06876=1195.356,-28.559,-42.395,179.889,5.628,149.026
C06877=1195.361,-28.808,-42.383,179.886,5.628,149.027
C06878=1195.366,-29.058,-42.371,179.884,5.627,149.027
C06879=1195.371,-29.308,-42.358,179.882,5.627,149.028
C06880=1195.376,-29.557,-42.345,179.879,5.627,149.028
C06881=1195.381,-29.806,-42.333,179.877,5.626,149.029
C06882=1195.386,-30.056,-42.320,179.874,5.626,149.030
C06883=1195.392,-30.306,-42.307,179.871,5.625,149.031
C06884=1195.397,-30.556,-42.295,179.869,5.626,149.031
C06885=1195.402,-30.805,-42.282,179.867,5.625,149.032
C06886=1195.407,-31.055,-42.269,179.864,5.624,149.032
C06887=1195.412,-31.304,-42.257,179.862,5.624,149.033
C06888=1195.417,-31.555,-42.245,179.860,5.624,149.034
C06889=1195.422,-31.804,-42.232,179.857,5.624,149.035
C06890=1195.427,-32.053,-42.219,179.855,5.623,149.035
C06891=1195.433,-32.303,-42.207,179.852,5.622,149.036
C06892=1195.438,-32.553,-42.195,179.850,5.623,149.036
C06893=1195.442,-32.803,-42.182,179.847,5.622,149.037
C06894=1195.448,-33.052,-42.169,179.845,5.622,149.038
C06895=1195.453,-33.302,-42.156,179.843,5.621,149.038
C06896=1195.459,-33.551,-42.144,179.841,5.621,149.039
C06897=1195.464,-33.801,-42.132,179.838,5.621,149.040
C06898=1195.469,-34.050,-42.119,179.835,5.620,149.040
C06899=1195.474,-34.301,-42.107,179.833,5.620,149.041
C06900=1195.479,-34.550,-42.094,179.830,5.619,149.042
C06901=1195.484,-34.799,-42.082,179.828,5.620,149.042
C06902=1195.490,-35.049,-42.070,179.826,5.619,149.043
C06903=1195.495,-35.299,-42.057,179.823,5.619,149.044
C06904=1195.500,-35.548,-42.045,179.820,5.618,149.044
C06905=1195.505,-35.798,-42.033,179.819,5.618,149.045
C06906=1195.510,-36.048,-42.020,179.816,5.618,149.045
C06907=1195.515,-36.297,-42.007,179.813,5.617,149.046
C06908=1195.520,-36.547,-41.995,179.811,5.618,149.047
C06909=1195.526,-36.796,-41.983,179.809,5.617,149.048
C06910=1195.531,-37.046,-41.971,179.806,5.616,149.048
C06911=1195.536,-37.296,-41.958,179.804,5.616,149.049
C06912=1195.541,-37.545,-41.946,179.802,5.616,149.049
C06913=1195.547,-37.795,-41.934,179.799,5.616,149.050
C06914=1195.551,-38.045,-41.921,179.796,5.615,149.051
C06915=1195.557,-38.295,-41.909,179.794,5.614,149.051
C06916=1195.562,-38.544,-41.896,179.792,5.615,149.052
C06917=1195.567,-38.794,-41.884,179.790,5.614,149.053
C06918=1195.571,-39.043,-41.872,179.787,5.614,149.053
C06919=1195.577,-39.293,-41.860,179.784,5.613,149.054
C06920=1195.582,-39.542,-41.848,179.783,5.613,149.055
C06921=1195.587,-39.792,-41.835,179.780,5.613,149.055
C06922=1195.593,-40.042,-41.823,179.777,5.612,149.056
C06923=1195.598,-40.291,-41.811,179.775,5.612,149.057
C06924=1195.603,-40.541,-41.799,179.773,5.612,149.057
C06925=1195.608,-40.790,-41.786,179.770,5.612,149.058
C06926=1195.613,-41.041,-41.774,179.768,5.611,149.059
C06927=1195.618,-41.290,-41.761,179.766,5.611,149.059
C06928=1195.623,-41.540,-41.750,179.763,5.611,149.060
C06929=1195.628,-41.790,-41.738,179.760,5.611,149.061
C06930=1195.633,-42.039,-41.726,179.758,5.610,149.061
C06931=1195.639,-42.289,-41.714,179.756,5.610,149.062
C06932=1195.644,-42.538,-41.701,179.753,5.610,149.063
C06933=1195.649,-42.788,-41.689,179.751,5.609,149.063
C06934=1195.655,-43.038,-41.677,179.748,5.609,149.064
C06935=1195.659,-43.287,-41.665,179.746,5.609,149.064
C06936=1195.664,-43.537,-41.653,179.744,5.608,149.065
C06937=1195.670,-43.786,-41.641,179.741,5.608,149.066
C06938=1195.675,-44.036,-41.629,179.739,5.608,149.067
C06939=1195.680,-44.286,-41.616,179.736,5.608,149.067
C06940=1195.686,-44.536,-41.605,179.734,5.607,149.068
C06941=1195.691,-44.785,-41.593,179.732,5.606,149.068
C06942=1195.696,-45.035,-41.581,179.729,5.607,149.069
C06943=1195.701,-45.285,-41.569,179.727,5.606,149.070
C06944=1195.706,-45.534,-41.556,179.724,5.606,149.071
C06945=1195.712,-45.784,-41.544,179.723,5.606,149.071
C06946=1195.716,-46.033,-41.533,179.720,5.605,149.072
C06947=1195.721,-46.283,-41.520,179.717,5.605,149.072
C06948=1195.727,-46.533,-41.508,179.715,5.604,149.073
C06949=1195.732,-46.783,-41.497,179.712,5.605,149.074
C06950=1195.737,-47.032,-41.485,179.710,5.604,149.074
C06951=1195.742,-47.282,-41.473,179.708,5.604,149.075
C06952=1195.748,-47.532,-41.461,179.706,5.604,149.076
C06953=1195.753,-47.781,-41.449,179.703,5.603,149.076
C06954=1195.757,-48.030,-41.437,179.700,5.603,149.077
C06955=1195.763,-48.280,-41.425,179.699,5.603,149.078
C06956=1195.768,-48.530,-41.413,179.696,5.603,149.078
C06957=1195.774,-48.780,-41.401,179.693,5.602,149.079
C06958=1195.780,-49.050,-41.389,179.691,5.602,149.080
C06959=1195.785,-49.320,-41.376,179.689,5.602,149.080
C06960=1195.790,-49.591,-41.363,179.686,5.602,149.081
C06961=1195.796,-49.860,-41.350,179.683,5.601,149.082
C06962=1195.802,-50.110,-41.338,179.680,5.601,149.082
C06963=1195.806,-50.359,-41.326,179.678,5.600,149.083
C06964=1195.811,-50.609,-41.314,179.676,5.600,149.084
C06965=1195.817,-50.859,-41.302,179.674,5.600,149.084
C06966=1195.821,-51.109,-41.291,179.671,5.599,149.085
C06967=1195.827,-51.359,-41.279,179.669,5.600,149.086
C06968=1195.832,-51.608,-41.267,179.666,5.599,149.086
C06969=1195.837,-51.858,-41.255,179.664,5.598,149.087
C06970=1195.842,-52.108,-41.244,179.662,5.599,149.088
C06971=1195.848,-52.357,-41.232,179.659,5.598,149.088
C06972=1195.853,-52.606,-41.221,179.657,5.598,149.089
C06973=1195.858,-52.856,-41.209,179.654,5.598,149.090
C06974=1195.864,-53.106,-41.197,179.652,5.597,149.090
C06975=1195.868,-53.355,-41.185,179.650,5.597,149.091
C06976=1195.874,-53.605,-41.173,179.648,5.597,149.092
C06977=1195.878,-53.855,-41.162,179.645,5.597,149.092
C06978=1195.884,-54.105,-41.150,179.643,5.596,149.093
C06979=1195.889,-54.355,-41.138,179.641,5.596,149.094
C06980=1195.894,-54.604,-41.127,179.638,5.596,149.094
C06981=1195.899,-54.854,-41.115,179.635,5.596,149.095
C06982=1195.904,-55.103,-41.104,179.633,5.595,149.096
C06983=1195.910,-55.353,-41.092,179.631,5.595,149.096
C06984=1195.915,-55.603,-41.080,179.628,5.595,149.097
C06985=1195.920,-55.853,-41.069,179.626,5.594,149.098
C06986=1195.925,-56.103,-41.057,179.624,5.595,149.098
C06987=1195.930,-56.352,-41.046,179.621,5.594,149.099
C06988=1195.936,-56.602,-41.034,179.619,5.593,149.099
C06989=1195.941,-56.851,-41.023,179.617,5.594,149.100
C06990=1195.946,-57.101,-41.011,179.614,5.593,149.101
C06991=1195.951,-57.351,-41.000,179.611,5.593,149.102
C06992=1195.956,-57.601,-40.988,179.610,5.593,149.102
C06993=1195.961,-57.850,-40.976,179.607,5.592,149.103
C06994=1195.967,-58.100,-40.965,179.604,5.592,149.103
C06995=1195.973,-58.349,-40.953,179.602,5.592,149.104
C06996=1195.977,-58.599,-40.942,179.600,5.592,149.105
C06997=1195.983,-58.849,-40.930,179.597,5.591,149.105
C06998=1195.987,-59.099,-40.919,179.595,5.591,149.106
C06999=1195.993,-59.349,-40.907,179.593,5.591,149.107
C07000=1195.998,-59.598,-40.895,179.591,5.591,149.107
C07001=1196.004,-59.847,-40.884,179.588,5.590,149.108
C07002=1196.008,-60.097,-40.873,179.586,5.590,149.109
C07003=1196.013,-60.347,-40.861,179.584,5.590,149.109
C07004=1196.018,-60.597,-40.849,179.581,5.590,149.110
C07005=1196.023,-60.846,-40.838,179.578,5.589,149.111
C07006=1196.029,-61.095,-40.827,179.577,5.589,149.111
C07007=1196.034,-61.345,-40.815,179.574,5.589,149.112
C07008=1196.040,-61.596,-40.804,179.571,5.589,149.113
C07009=1196.044,-61.845,-40.793,179.569,5.589,149.113
C07010=1196.050,-62.094,-40.781,179.567,5.588,149.114
C07011=1196.055,-62.344,-40.770,179.565,5.588,149.114
C07012=1196.060,-62.594,-40.758,179.562,5.588,149.115
C07013=1196.065,-62.844,-40.747,179.560,5.588,149.116
C07014=1196.070,-63.093,-40.736,179.557,5.587,149.117
C07015=1196.076,-63.343,-40.725,179.556,5.587,149.117
C07016=1196.081,-63.593,-40.714,179.553,5.587,149.118
C07017=1196.086,-63.843,-40.702,179.550,5.586,149.118
C07018=1196.091,-64.092,-40.691,179.548,5.587,149.119
C07019=1196.096,-64.341,-40.679,179.546,5.586,149.120
C07020=1196.102,-64.592,-40.668,179.544,5.586,149.120
C07021=1196.107,-64.841,-40.657,179.541,5.586,149.121
C07022=1196.113,-65.091,-40.645,179.538,5.585,149.122
C07023=1196.117,-65.340,-40.634,179.536,5.586,149.122
C07024=1196.122,-65.590,-40.623,179.534,5.585,149.123
C07025=1196.128,-65.841,-40.612,179.532,5.584,149.124
C07026=1196.133,-66.089,-40.601,179.529,5.585,149.124
C07027=1196.138,-66.339,-40.589,179.527,5.584,149.125
C07028=1196.143,-66.589,-40.578,179.525,5.584,149.126
C07029=1196.149,-66.839,-40.567,179.523,5.584,149.126
C07030=1196.154,-67.088,-40.556,179.520,5.584,149.127
C07031=1196.159,-67.338,-40.544,179.518,5.584,149.128
C07032=1196.164,-67.588,-40.534,179.516,5.583,149.128
C07033=1196.170,-67.838,-40.522,179.513,5.583,149.129
C07034=1196.175,-68.087,-40.511,179.511,5.583,149.130
C07035=1196.180,-68.337,-40.500,179.508,5.583,149.130
C07036=1196.185,-68.586,-40.489,179.506,5.582,149.131
C07037=1196.190,-68.836,-40.477,179.504,5.582,149.131
C07038=1196.195,-69.086,-40.466,179.501,5.582,149.132
C07039=1196.201,-69.335,-40.456,179.499,5.582,149.133
C07040=1196.206,-69.585,-40.444,179.497,5.582,149.134
C07041=1196.211,-69.836,-40.433,179.494,5.581,149.134
C07042=1196.216,-70.085,-40.423,179.492,5.581,149.135
C07043=1196.222,-70.335,-40.411,179.490,5.581,149.135
C07044=1196.227,-70.585,-40.400,179.487,5.580,149.136
C07045=1196.232,-70.834,-40.389,179.485,5.580,149.137
C07046=1196.237,-71.083,-40.378,179.483,5.580,149.137
C07047=1196.243,-71.333,-40.367,179.481,5.580,149.138
C07048=1196.248,-71.583,-40.356,179.478,5.580,149.139
C07049=1196.253,-71.833,-40.345,179.476,5.579,149.139
C07050=1196.258,-72.082,-40.334,179.474,5.579,149.140
C07051=1196.264,-72.333,-40.323,179.471,5.579,149.141
C07052=1196.268,-72.582,-40.312,179.469,5.579,149.141
C07053=1196.274,-72.831,-40.301,179.467,5.579,149.142
C07054=1196.279,-73.081,-40.290,179.464,5.578,149.143
C07055=1196.285,-73.331,-40.279,179.462,5.579,149.143
C07056=1196.290,-73.581,-40.268,179.459,5.578,149.144
C07057=1196.294,-73.830,-40.257,179.457,5.577,149.144
C07058=1196.300,-74.080,-40.247,179.455,5.578,149.145
C07059=1196.305,-74.330,-40.235,179.452,5.577,149.146
C07060=1196.311,-74.579,-40.225,179.450,5.578,149.147
C07061=1196.316,-74.829,-40.213,179.448,5.577,149.147
C07062=1196.321,-75.100,-40.201,179.445,5.576,149.148
C07063=1196.327,-75.371,-40.191,179.443,5.577,149.148
C07064=1196.333,-75.642,-40.178,179.441,5.576,149.149
C07065=1196.338,-75.913,-40.166,179.438,5.576,149.150
C07066=1196.344,-76.162,-40.156,179.435,5.575,149.151
C07067=1196.349,-76.412,-40.145,179.433,5.576,149.151
C07068=1196.354,-76.661,-40.134,179.431,5.575,149.152
C07069=1196.359,-76.911,-40.123,179.429,5.575,149.153
C07070=1196.365,-77.160,-40.113,179.426,5.575,149.153
C07071=1196.370,-77.410,-40.101,179.424,5.575,149.154
C07072=1196.376,-77.660,-40.091,179.421,5.575,149.155
C07073=1196.381,-77.910,-40.080,179.419,5.574,149.155
C07074=1196.385,-78.160,-40.069,179.417,5.574,149.156
C07075=1196.391,-78.409,-40.059,179.415,5.574,149.157
C07076=1196.396,-78.659,-40.047,179.412,5.573,149.157
C07077=1196.401,-78.909,-40.037,179.410,5.574,149.158
C07078=1196.406,-79.159,-40.027,179.408,5.573,149.158
C07079=1196.412,-79.408,-40.016,179.406,5.574,149.159
C07080=1196.417,-79.658,-40.005,179.403,5.573,149.160
C07081=1196.423,-79.907,-39.994,179.401,5.573,149.160
C07082=1196.428,-80.157,-39.983,179.399,5.573,149.161
C07083=1196.433,-80.407,-39.973,179.396,5.572,149.162
C07084=1196.438,-80.657,-39.962,179.394,5.572,149.162
C07085=1196.443,-80.906,-39.951,179.392,5.572,149.163
C07086=1196.448,-81.156,-39.941,179.390,5.572,149.164
C07087=1196.454,-81.405,-39.930,179.387,5.572,149.164
C07088=1196.459,-81.656,-39.919,179.385,5.571,149.165
C07089=1196.464,-81.905,-39.909,179.383,5.571,149.166
C07090=1196.469,-82.155,-39.898,179.380,5.571,149.166
C07091=1196.475,-82.404,-39.888,179.378,5.571,149.167
C07092=1196.480,-82.655,-39.877,179.376,5.571,149.167
C07093=1196.485,-82.904,-39.867,179.374,5.571,149.168
C07094=1196.490,-83.154,-39.855,179.371,5.571,149.169
C07095=1196.495,-83.403,-39.845,179.369,5.570,149.169
C07096=1196.500,-83.653,-39.835,179.367,5.570,149.170
C07097=1196.506,-83.903,-39.824,179.364,5.570,149.171
C07098=1196.511,-84.153,-39.813,179.362,5.570,149.171
C07099=1196.516,-84.402,-39.803,179.360,5.569,149.172
C07100=1196.521,-84.652,-39.792,179.357,5.569,149.173
C07101=1196.527,-84.902,-39.782,179.355,5.569,149.173
C07102=1196.532,-85.152,-39.771,179.352,5.569,149.174
C07103=1196.537,-85.401,-39.761,179.351,5.569,149.175
C07104=1196.542,-85.651,-39.750,179.348,5.568,149.175
C07105=1196.548,-85.901,-39.740,179.346,5.569,149.176
C07106=1196.553,-86.150,-39.730,179.344,5.568,149.176
C07107=1196.558,-86.401,-39.719,179.341,5.568,149.177
C07108=1196.564,-86.650,-39.708,179.339,5.568,149.178
C07109=1196.569,-86.900,-39.698,179.336,5.567,149.179
C07110=1196.574,-87.149,-39.687,179.335,5.567,149.179
C07111=1196.579,-87.400,-39.677,179.332,5.567,149.180
C07112=1196.585,-87.649,-39.667,179.330,5.567,149.180
C07113=1196.590,-87.899,-39.656,179.328,5.567,149.181
C07114=1196.594,-88.148,-39.646,179.326,5.567,149.182
C07115=1196.600,-88.398,-39.635,179.323,5.567,149.182
C07116=1196.605,-88.648,-39.625,179.320,5.566,149.183
C07117=1196.611,-88.897,-39.615,179.319,5.566,149.184
C07118=1196.616,-89.148,-39.604,179.316,5.566,149.184
C07119=1196.621,-89.397,-39.594,179.314,5.566,149.185
C07120=1196.627,-89.647,-39.584,179.312,5.565,149.185
C07121=1196.632,-89.897,-39.573,179.310,5.566,149.186
C07122=1196.637,-90.147,-39.563,179.307,5.565,149.187
C07123=1196.642,-90.397,-39.552,179.304,5.565,149.188
C07124=1196.647,-90.645,-39.542,179.303,5.565,149.188
C07125=1196.653,-90.895,-39.532,179.300,5.565,149.189
C07126=1196.658,-91.145,-39.521,179.298,5.565,149.190
C07127=1196.663,-91.395,-39.511,179.296,5.564,149.190
C07128=1196.669,-91.644,-39.501,179.294,5.564,149.191
C07129=1196.674,-91.895,-39.490,179.291,5.564,149.191
C07130=1196.679,-92.144,-39.480,179.289,5.564,149.192
C07131=1196.684,-92.394,-39.470,179.287,5.564,149.193
C07132=1196.689,-92.644,-39.460,179.285,5.564,149.193
C07133=1196.695,-92.893,-39.450,179.282,5.564,149.194
C07134=1196.700,-93.143,-39.439,179.280,5.563,149.195
C07135=1196.705,-93.393,-39.429,179.278,5.563,149.195
C07136=1196.710,-93.642,-39.419,179.275,5.563,149.196
C07137=1196.715,-93.892,-39.409,179.273,5.563,149.196
C07138=1196.721,-94.142,-39.398,179.271,5.562,149.197
C07139=1196.727,-94.391,-39.388,179.269,5.563,149.198
C07140=1196.732,-94.642,-39.378,179.267,5.562,149.198
C07141=1196.736,-94.891,-39.368,179.264,5.562,149.199
C07142=1196.742,-95.140,-39.358,179.262,5.562,149.200
C07143=1196.747,-95.391,-39.348,179.259,5.562,149.200
C07144=1196.753,-95.641,-39.338,179.258,5.562,149.201
C07145=1196.758,-95.890,-39.328,179.255,5.561,149.202
C07146=1196.763,-96.140,-39.318,179.253,5.562,149.202
C07147=1196.768,-96.390,-39.307,179.251,5.561,149.203
C07148=1196.774,-96.639,-39.297,179.248,5.561,149.204
C07149=1196.780,-96.889,-39.287,179.246,5.561,149.204
C07150=1196.784,-97.139,-39.277,179.244,5.561,149.205
C07151=1196.789,-97.388,-39.267,179.242,5.560,149.205
C07152=1196.795,-97.638,-39.257,179.239,5.561,149.206
C07153=1196.800,-97.889,-39.247,179.237,5.560,149.207
C07154=1196.805,-98.138,-39.237,179.235,5.560,149.207
C07155=1196.811,-98.388,-39.227,179.232,5.560,149.208
C07156=1196.816,-98.637,-39.217,179.230,5.559,149.209
C07157=1196.821,-98.887,-39.207,179.228,5.559,149.209
C07158=1196.826,-99.137,-39.197,179.226,5.559,149.210
C07159=1196.832,-99.387,-39.187,179.224,5.559,149.211
C07160=1196.838,-99.636,-39.177,179.221,5.559,149.211
C07161=1196.842,-99.886,-39.167,179.219,5.559,149.212
C07162=1196.848,-100.136,-39.157,179.216,5.559,149.213
C07163=1196.853,-100.385,-39.146,179.215,5.559,149.213
C07164=1196.858,-100.635,-39.137,179.212,5.558,149.214
C07165=1196.863,-100.885,-39.127,179.210,5.559,149.215
C07166=1196.869,-101.156,-39.116,179.208,5.558,149.215
C07167=1196.875,-101.428,-39.105,179.205,5.557,149.216
C07168=1196.881,-101.700,-39.095,179.203,5.558,149.216
C07169=1196.886,-101.971,-39.084,179.200,5.557,149.217
C07170=1196.891,-102.220,-39.073,179.198,5.558,149.218
C07171=1196.897,-102.471,-39.064,179.196,5.557,149.219
C07172=1196.902,-102.720,-39.054,179.194,5.557,149.219
C07173=1196.907,-102.970,-39.044,179.191,5.557,149.220
C07174=1196.912,-103.219,-39.034,179.189,5.556,149.220
C07175=1196.918,-103.469,-39.025,179.187,5.557,149.221
C07176=1196.923,-103.719,-39.014,179.185,5.556,149.222
C07177=1196.928,-103.968,-39.005,179.183,5.556,149.222
C07178=1196.934,-104.219,-38.995,179.180,5.556,149.223
C07179=1196.939,-104.469,-38.985,179.178,5.556,149.224
C07180=1196.944,-104.718,-38.975,179.176,5.555,149.224
C07181=1196.950,-104.968,-38.966,179.174,5.556,149.225
C07182=1196.955,-105.217,-38.956,179.171,5.555,149.226
C07183=1196.960,-105.468,-38.945,179.170,5.555,149.226
C07184=1196.965,-105.717,-38.937,179.167,5.555,149.227
C07185=1196.971,-105.967,-38.926,179.165,5.555,149.227
C07186=1196.976,-106.216,-38.916,179.163,5.555,149.228
C07187=1196.981,-106.466,-38.907,179.161,5.555,149.229
C07188=1196.986,-106.717,-38.897,179.158,5.555,149.229
C07189=1196.991,-106.966,-38.887,179.156,5.555,149.230
C07190=1196.997,-107.216,-38.878,179.154,5.554,149.231
C07191=1197.002,-107.465,-38.868,179.152,5.555,149.231
C07192=1197.008,-107.715,-38.858,179.149,5.554,149.232
C07193=1197.013,-107.965,-38.849,179.147,5.554,149.232
C07194=1197.018,-108.215,-38.838,179.145,5.554,149.233
C07195=1197.023,-108.465,-38.829,179.143,5.554,149.234
C07196=1197.029,-108.714,-38.819,179.140,5.553,149.234
C07197=1197.034,-108.964,-38.810,179.138,5.554,149.235
C07198=1197.039,-109.214,-38.800,179.136,5.553,149.236
C07199=1197.044,-109.463,-38.791,179.134,5.553,149.236
C07200=1197.050,-109.713,-38.781,179.132,5.553,149.237
C07201=1197.055,-109.962,-38.771,179.130,5.553,149.238
C07202=1197.060,-110.213,-38.762,179.127,5.553,149.238
C07203=1197.065,-110.462,-38.752,179.125,5.553,149.239
C07204=1197.071,-110.712,-38.742,179.123,5.552,149.239
C07205=1197.076,-110.962,-38.733,179.121,5.553,149.240
C07206=1197.082,-111.212,-38.723,179.118,5.552,149.241
C07207=1197.087,-111.461,-38.714,179.116,5.552,149.241
C07208=1197.093,-111.711,-38.704,179.114,5.552,149.242
C07209=1197.097,-111.960,-38.695,179.112,5.552,149.243
C07210=1197.103,-112.211,-38.685,179.109,5.551,149.243
C07211=1197.108,-112.461,-38.675,179.108,5.551,149.244
C07212=1197.113,-112.711,-38.666,179.105,5.551,149.244
C07213=1197.118,-112.960,-38.656,179.103,5.551,149.245
C07214=1197.123,-113.210,-38.647,179.101,5.551,149.246
C07215=1197.129,-113.459,-38.637,179.099,5.551,149.246
C07216=1197.134,-113.709,-38.628,179.096,5.551,149.247
C07217=1197.140,-113.959,-38.618,179.094,5.551,149.248
C07218=1197.145,-114.209,-38.609,179.092,5.550,149.248
C07219=1197.151,-114.459,-38.599,179.090,5.550,149.249
C07220=1197.156,-114.708,-38.590,179.087,5.550,149.249
C07221=1197.161,-114.958,-38.581,179.085,5.550,149.250
C07222=1197.167,-115.208,-38.571,179.083,5.549,149.251
C07223=1197.172,-115.457,-38.562,179.081,5.550,149.251
C07224=1197.178,-115.707,-38.552,179.079,5.549,149.252
C07225=1197.182,-115.957,-38.542,179.077,5.549,149.253
C07226=1197.187,-116.207,-38.533,179.074,5.549,149.253
C07227=1197.193,-116.457,-38.524,179.073,5.549,149.254
C07228=1197.198,-116.707,-38.514,179.070,5.549,149.255
C07229=1197.203,-116.956,-38.505,179.068,5.549,149.255
C07230=1197.209,-117.206,-38.495,179.066,5.548,149.256
C07231=1197.214,-117.456,-38.486,179.064,5.549,149.256
C07232=1197.220,-117.706,-38.477,179.061,5.548,149.257
C07233=1197.224,-117.955,-38.467,179.059,5.548,149.258
C07234=1197.230,-118.205,-38.458,179.057,5.548,149.258
C07235=1197.236,-118.455,-38.449,179.055,5.548,149.259
C07236=1197.240,-118.704,-38.439,179.052,5.548,149.260
C07237=1197.246,-118.954,-38.430,179.051,5.548,149.260
C07238=1197.251,-119.204,-38.421,179.048,5.547,149.261
C07239=1197.257,-119.454,-38.412,179.046,5.548,149.261
C07240=1197.262,-119.704,-38.402,179.044,5.547,149.262
C07241=1197.267,-119.953,-38.393,179.042,5.547,149.263
C07242=1197.273,-120.204,-38.384,179.040,5.547,149.263
C07243=1197.277,-120.453,-38.374,179.037,5.547,149.264
C07244=1197.283,-120.703,-38.365,179.035,5.547,149.265
C07245=1197.289,-120.953,-38.356,179.033,5.546,149.265
C07246=1197.294,-121.203,-38.347,179.031,5.547,149.266
C07247=1197.299,-121.452,-38.337,179.029,5.546,149.266
C07248=1197.304,-121.702,-38.328,179.027,5.546,149.267
C07249=1197.310,-121.952,-38.319,179.024,5.546,149.268
C07250=1197.315,-122.202,-38.310,179.022,5.546,149.268
C07251=1197.320,-122.452,-38.301,179.020,5.546,149.269
C07252=1197.325,-122.701,-38.292,179.018,5.546,149.269
C07253=1197.331,-122.951,-38.282,179.015,5.545,149.270
C07254=1197.336,-123.201,-38.273,179.014,5.545,149.271
C07255=1197.341,-123.451,-38.264,179.011,5.545,149.271
C07256=1197.346,-123.701,-38.255,179.009,5.545,149.272
C07257=1197.352,-123.950,-38.245,179.007,5.545,149.273
C07258=1197.358,-124.199,-38.237,179.005,5.545,149.273
C07259=1197.363,-124.449,-38.228,179.003,5.544,149.274
C07260=1197.368,-124.699,-38.219,179.001,5.545,149.274
C07261=1197.374,-124.949,-38.209,178.999,5.545,149.275
C07262=1197.379,-125.199,-38.200,178.996,5.544,149.276
C07263=1197.384,-125.448,-38.191,178.994,5.545,149.276
C07264=1197.389,-125.698,-38.182,178.992,5.544,149.277
C07265=1197.394,-125.948,-38.173,178.990,5.544,149.278
C07266=1197.399,-126.198,-38.164,178.988,5.543,149.278
C07267=1197.405,-126.448,-38.155,178.986,5.544,149.279
C07268=1197.410,-126.698,-38.146,178.983,5.543,149.279
C07269=1197.416,-126.948,-38.137,178.981,5.543,149.280
C07270=1196.994,-126.959,-38.176,178.977,5.547,149.282
C07271=1196.989,-126.709,-38.185,178.979,5.547,149.281
C07272=1196.984,-126.459,-38.193,178.982,5.547,149.281
C07273=1196.978,-126.209,-38.203,178.983,5.547,149.280
C07274=1196.973,-125.959,-38.212,178.986,5.547,149.279
C07275=1196.968,-125.709,-38.221,178.988,5.547,149.279
C07276=1196.963,-125.459,-38.230,178.990,5.548,149.278
C07277=1196.957,-125.209,-38.238,178.992,5.547,149.278
C07278=1196.951,-124.959,-38.248,178.995,5.548,149.277
C07279=1196.947,-124.710,-38.258,178.997,5.548,149.276
C07280=1196.941,-124.461,-38.266,178.999,5.549,149.276
C07281=1196.936,-124.211,-38.275,179.001,5.548,149.275
C07282=1196.931,-123.961,-38.284,179.003,5.548,149.274
C07283=1196.925,-123.711,-38.293,179.005,5.548,149.274
C07284=1196.919,-123.461,-38.302,179.007,5.548,149.273
C07285=1196.915,-123.212,-38.312,179.009,5.549,149.273
C07286=1196.909,-122.962,-38.321,179.012,5.548,149.272
C07287=1196.904,-122.712,-38.330,179.014,5.549,149.271
C07288=1196.898,-122.462,-38.339,179.016,5.549,149.271
C07289=1196.893,-122.212,-38.348,179.019,5.549,149.270
C07290=1196.888,-121.963,-38.358,179.020,5.549,149.270
C07291=1196.882,-121.713,-38.367,179.023,5.550,149.269
C07292=1196.877,-121.463,-38.376,179.024,5.550,149.268
C07293=1196.872,-121.213,-38.385,179.027,5.550,149.268
C07294=1196.867,-120.964,-38.395,179.029,5.550,149.267
C07295=1196.861,-120.714,-38.404,179.031,5.550,149.266
C07296=1196.856,-120.464,-38.413,179.033,5.550,149.266
C07297=1196.851,-120.214,-38.422,179.036,5.551,149.265
C07298=1196.845,-119.964,-38.432,179.038,5.550,149.265
C07299=1196.840,-119.715,-38.441,179.040,5.551,149.264
C07300=1196.835,-119.465,-38.450,179.042,5.551,149.263
C07301=1196.830,-119.215,-38.460,179.045,5.551,149.263
C07302=1196.824,-118.965,-38.469,179.046,5.551,149.262
C07303=1196.819,-118.715,-38.478,179.048,5.551,149.261
C07304=1196.814,-118.466,-38.487,179.051,5.552,149.261
C07305=1196.808,-118.216,-38.497,179.053,5.551,149.260
C07306=1196.803,-117.966,-38.506,179.055,5.551,149.259
